KUKA KRL program: Vessel04speedt3.src

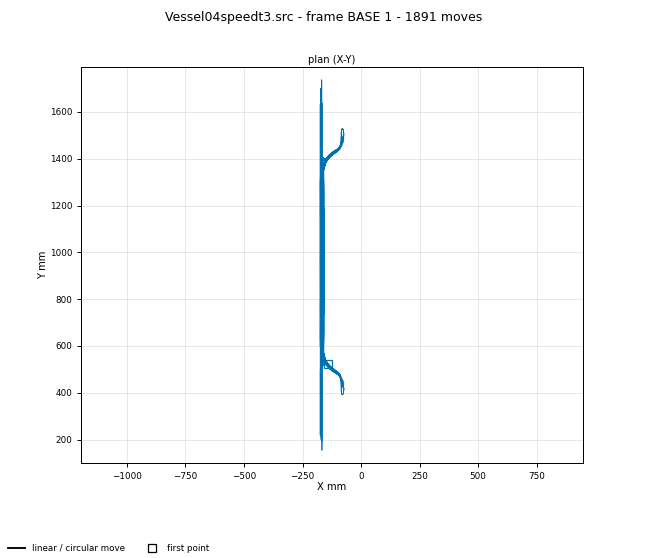
[picture p0: tool path of Vessel04speedt3.src in frame BASE 1, 1891 of 1892 moves have a stored position in this frame; points joined in program order, loops and branches not executed]
&ACCESS RVP
DEF Vessel_04( )
;FOLD INI;%{PE}%V2.2.2,%MKUKATPBASIS,%CINIT,%VCOMMON,%P
;FOLD BAS INI;%{PE}%V2.2.2,%MKUKATPBASIS,%CINIT,%VINIT,%P
INTERRUPT DECL 3 WHEN $STOPMESS==TRUE DO IR_STOPM ( )
INTERRUPT ON 3
BAS (#INITMOV,0 )
;ENDFOLD
;FOLD USER INI;%{P}%V2.2.2,%MKUKATPUSER,%CINIT,%VINIT,%P
;Make your modifications here

;ENDFOLD
;ENDFOLD
ACTION(#AXIS_RESET,34,1000,#NOERROR,ERROR_CODE)
;FOLD PTP HOME  Vel= 100 % DEFAULT;%{PE}%V2.2.2,%MKUKATPBASIS,%CMOVE,%VPTP,%P 1:PTP, 2:HOME, 3:, 5:100, 7:DEFAULT
$H_POS=XHOME
PDAT_ACT=PDEFAULT
BAS (#PTP_DAT )
FDAT_ACT=FHOME
BAS (#FRAMES )
BAS (#VEL_PTP,100 )
PTP  XHOME
;ENDFOLD
BAS(#TOOL,1)
BAS(#BASE,1)
LIN {X -141.371,Y 523.534,Z 0.000,A 30.000, B 0.00, C 0.00,E1 -59.199}
HALT

; PLY 1 OF 41 (Helical)

; ANGLE 51.0 (Not valid for Circ layers and non-tubes)
$APO.CDIS=85
$VEL_EXTAX[1]=100
FOR N_CYC=1 to 56
 LIN_REL {X  -10.568,Y +19.006,A +0.000,E1 -7.240,E3 +6.829,E4 +6.829} C_DIS
 LIN_REL {X  -10.476,Y +36.643,A +0.000,E1 -6.561,E3 +10.073,E4 +10.073} C_DIS
 LIN_REL {X  -2.489,Y +48.216,A -0.000,E1 -2.729,E3 +13.363,E4 +13.363} C_DIS
 LIN_REL {X  +0.199,Y +33.447,A -2.982,E1 -0.404,E3 +10.273,E4 +10.273} C_DIS
 LIN_REL {X  +0.568,Y +37.624,A -7.584,E1 -0.184,E3 +12.184,E4 +12.184} C_DIS
 LIN_REL {X  +1.054,Y +53.527,A -6.791,E1 -0.176,E3 +18.278,E4 +18.278} C_DIS
 LIN_REL {X  +0.629,Y +62.690,A -5.877,E1 +0.690,E3 +22.592,E4 +22.592} C_DIS
 LIN_REL {X  -0.282,Y +46.012,A -4.843,E1 +0.643,E3 +17.284,E4 +17.284} C_DIS
 LIN_REL {X  -0.828,Y +43.828,A -1.901,E1 +0.054,E3 +17.077,E4 +17.077} C_DIS
 LIN_REL {X  -0.963,Y +65.510,A -0.022,E1 -0.470,E3 +27.232,E4 +27.232} C_DIS
 LIN_REL {X  +0.036,Y +73.951,A +0.000,E1 +0.019,E3 +32.052,E4 +32.052} C_DIS
 LIN_REL {X  +0.003,Y +169.509,A +0.000,E1 +0.001,E3 +73.597,E4 +73.597} C_DIS
 LIN_REL {X  +0.150,Y +71.344,A +0.000,E1 +0.017,E3 +31.107,E4 +31.107} C_DIS
 LIN_REL {X  +3.036,Y +57.808,A +0.000,E1 +0.283,E3 +27.550,E4 +27.550} C_DIS
 LIN_REL {X  +11.901,Y +41.351,A +0.000,E1 +1.145,E3 +26.975,E4 +26.975} C_DIS
 LIN_REL {X  +17.652,Y +24.337,A -0.003,E1 +1.971,E3 +20.974,E4 +20.974} C_DIS
 LIN_REL {X  +10.669,Y +8.551,A -2.858,E1 +1.178,E3 +8.021,E4 +8.021} C_DIS
 LIN_REL {X  +17.182,Y +15.853,A -9.749,E1 +3.486,E3 +17.744,E4 +17.744} C_DIS
 LIN_REL {X  +18.322,Y +27.598,A -9.305,E1 +5.329,E3 +37.822,E4 +37.822} C_DIS
 LIN_REL {X  +8.849,Y +21.653,A -6.390,E1 +5.112,E3 +38.276,E4 +38.276} C_DIS
 LIN_REL {X  +4.056,Y +23.007,A -1.638,E1 +5.484,E3 +50.951,E4 +50.951} C_DIS
 LIN_REL {X  -4.096,Y +21.816,A -0.057,E1 +6.652,E3 +66.123,E4 +66.123} C_DIS
 LIN_REL {X  -5.666,Y +0.355,A +0.000,E1 +5.437,E3 +42.648,E4 +42.648} C_DIS
 LIN_REL {X  -2.099,Y -14.454,A +0.000,E1 +6.219,E3 +26.192,E4 +26.192} C_DIS
 LIN_REL {X  -0.280,Y -28.083,A +0.000,E1 +13.715,E3 +25.118,E4 +25.118} C_DIS
 LIN_REL {X  -0.395,Y -28.470,A +0.000,E1 +18.975,E3 +19.603,E4 +19.603} C_DIS
 LIN_REL {X  -9.197,Y -20.928,A +0.000,E1 +22.023,E3 +21.222,E4 +21.222} C_DIS
 LIN_REL {X  -19.997,Y -14.564,A +0.000,E1 +18.453,E3 +20.224,E4 +20.224} C_DIS
 LIN_REL {X  -17.121,Y -13.356,A +0.000,E1 +14.454,E3 +11.101,E4 +11.101} C_DIS
 LIN_REL {X  -9.075,Y -8.563,A +0.000,E1 +4.448,E3 +5.875,E4 +5.875} C_DIS
 LIN_REL {X  -9.764,Y -16.650,A +0.000,E1 +6.452,E3 +6.408,E4 +6.408} C_DIS
 LIN_REL {X  -12.054,Y -40.028,A +0.000,E1 +7.722,E3 +11.062,E4 +11.062} C_DIS
 LIN_REL {X  -2.489,Y -48.280,A +0.000,E1 +2.729,E3 +13.364,E4 +13.364} C_DIS
 LIN_REL {X  +0.199,Y -33.492,A +2.982,E1 +0.404,E3 +10.272,E4 +10.272} C_DIS
 LIN_REL {X  +0.568,Y -37.669,A +7.584,E1 +0.184,E3 +12.184,E4 +12.184} C_DIS
 LIN_REL {X  +1.054,Y -53.586,A +6.791,E1 +0.176,E3 +18.279,E4 +18.279} C_DIS
 LIN_REL {X  +0.629,Y -62.759,A +5.877,E1 -0.690,E3 +22.592,E4 +22.592} C_DIS
 LIN_REL {X  -0.282,Y -46.062,A +4.843,E1 -0.643,E3 +17.283,E4 +17.283} C_DIS
 LIN_REL {X  -0.828,Y -43.872,A +1.901,E1 -0.054,E3 +17.077,E4 +17.077} C_DIS
 LIN_REL {X  -0.963,Y -65.584,A +0.022,E1 +0.470,E3 +27.232,E4 +27.232} C_DIS
 LIN_REL {X  +0.036,Y -74.040,A +0.000,E1 -0.019,E3 +32.053,E4 +32.053} C_DIS
 LIN_REL {X  +0.003,Y -169.741,A +0.000,E1 -0.001,E3 +73.597,E4 +73.597} C_DIS
 LIN_REL {X  +0.150,Y -71.439,A +0.000,E1 -0.017,E3 +31.106,E4 +31.106} C_DIS
 LIN_REL {X  +3.036,Y -57.877,A +0.000,E1 -0.283,E3 +27.551,E4 +27.551} C_DIS
 LIN_REL {X  +11.901,Y -41.410,A +0.000,E1 -1.145,E3 +26.974,E4 +26.974} C_DIS
 LIN_REL {X  +17.652,Y -24.387,A +0.003,E1 -1.971,E3 +20.974,E4 +20.974} C_DIS
 LIN_REL {X  +10.669,Y -8.581,A +2.858,E1 -1.178,E3 +8.021,E4 +8.021} C_DIS
 LIN_REL {X  +17.182,Y -15.882,A +9.749,E1 -3.486,E3 +17.745,E4 +17.745} C_DIS
 LIN_REL {X  +18.322,Y -27.638,A +9.305,E1 -5.329,E3 +37.822,E4 +37.822} C_DIS
 LIN_REL {X  +8.849,Y -21.682,A +6.390,E1 -5.112,E3 +38.276,E4 +38.276} C_DIS
 LIN_REL {X  +4.056,Y -23.042,A +1.638,E1 -5.484,E3 +50.950,E4 +50.950} C_DIS
 LIN_REL {X  -4.096,Y -21.856,A +0.057,E1 -6.652,E3 +66.124,E4 +66.124} C_DIS
 LIN_REL {X  -5.666,Y -0.329,A -0.000,E1 -5.437,E3 +42.647,E4 +42.647} C_DIS
 LIN_REL {X  -2.099,Y +14.582,A -0.000,E1 -6.219,E3 +26.193,E4 +26.193} C_DIS
 LIN_REL {X  -0.280,Y +28.321,A -0.000,E1 -13.715,E3 +25.117,E4 +25.117} C_DIS
 LIN_REL {X  -0.395,Y +28.733,A -0.000,E1 -18.975,E3 +19.604,E4 +19.604} C_DIS
 LIN_REL {X  -9.197,Y +21.087,A -0.000,E1 -22.023,E3 +21.222,E4 +21.222} C_DIS
 LIN_REL {X  -19.997,Y +14.748,A -0.000,E1 -18.452,E3 +20.222,E4 +20.222} C_DIS
 LIN_REL {X  -26.970,Y +23.197,A -0.000,E1 -19.276,E3 +17.546,E4 +17.546} C_DIS
ENDFOR

HALT
LIN {X -165.446,Y 526.668,Z 0.000,A 30.000, B 0.00, C 0.00,E1 -64.562}
HALT

; PLY 2 OF 41 (Connector)

; ANGLE 51.0 (Not valid for Circ layers and non-tubes)
$APO.CDIS=85
$VEL_EXTAX[1]=100
FOR N_CYC=1 to 1
 LIN_REL {X  +0.000,Y +6.669,A +0.000,E1 -1.453,E3 +1.289,E4 +1.289} C_DIS
 LIN_REL {X  +0.000,Y +15.761,A +0.000,E1 -3.190,E3 +3.934,E4 +3.934} C_DIS
 LIN_REL {X  +0.000,Y +31.342,A +0.000,E1 -3.400,E3 +9.789,E4 +9.789} C_DIS
 LIN_REL {X  +0.000,Y +43.799,A +0.000,E1 -1.567,E3 +14.926,E4 +14.926} C_DIS
 LIN_REL {X  +0.000,Y +28.255,A -1.983,E1 -0.087,E3 +10.643,E4 +10.643} C_DIS
 LIN_REL {X  +0.000,Y +29.952,A -7.476,E1 +0.318,E3 +11.872,E4 +11.872} C_DIS
 LIN_REL {X  +0.000,Y +47.685,A -7.690,E1 +0.225,E3 +20.095,E4 +20.095} C_DIS
 LIN_REL {X  +0.000,Y +55.129,A -7.422,E1 +0.668,E3 +25.472,E4 +25.472} C_DIS
 LIN_REL {X  +0.000,Y +43.863,A -4.702,E1 +1.177,E3 +22.727,E4 +22.727} C_DIS
 LIN_REL {X  +0.000,Y +50.043,A -0.726,E1 +1.544,E3 +40.796,E4 +40.796} C_DIS
 LIN_REL {X  +0.000,Y +46.945,A -0.001,E1 +3.695,E3 +57.103,E4 +57.103} C_DIS
 LIN_REL {X  +0.000,Y +58.316,A +0.000,E1 +4.226,E3 +72.975,E4 +72.975} C_DIS
 LIN_REL {X  +0.000,Y +65.060,A +0.000,E1 +4.740,E3 +89.502,E4 +89.502} C_DIS
 LIN_REL {X  +0.000,Y +67.059,A +0.000,E1 +5.237,E3 +105.894,E4 +105.894} C_DIS
 LIN_REL {X  +0.000,Y +54.897,A +0.000,E1 +4.784,E3 +101.231,E4 +101.231} C_DIS
 LIN_REL {X  +0.000,Y +40.560,A +0.000,E1 +3.986,E3 +86.611,E4 +86.611} C_DIS
 LIN_REL {X  +0.000,Y +28.994,A +0.000,E1 +3.229,E3 +70.429,E4 +70.429} C_DIS
 LIN_REL {X  +0.000,Y +20.924,A -0.000,E1 +3.270,E3 +56.833,E4 +56.833} C_DIS
 LIN_REL {X  +0.000,Y +10.940,A -0.000,E1 +2.663,E3 +31.936,E4 +31.936} C_DIS
 LIN_REL {X  +0.000,Y +9.716,A -0.000,E1 +1.163,E3 +31.606,E4 +31.606} C_DIS
 LIN_REL {X  +0.000,Y +17.235,A -0.000,E1 +1.953,E3 +55.180,E4 +55.180} C_DIS
 LIN_REL {X  +0.000,Y +19.045,A -0.003,E1 +3.492,E3 +73.663,E4 +73.663} C_DIS
 LIN_REL {X  +0.000,Y +14.681,A -0.050,E1 +3.224,E3 +66.879,E4 +66.879} C_DIS
 LIN_REL {X  +0.000,Y +9.269,A -0.348,E1 +2.308,E3 +46.823,E4 +46.823} C_DIS
 LIN_REL {X  +0.000,Y +6.944,A -1.216,E1 +1.589,E3 +34.534,E4 +34.534} C_DIS
 LIN_REL {X  +0.000,Y +4.516,A -2.642,E1 +2.440,E3 +22.764,E4 +22.764} C_DIS
 LIN_REL {X  +0.000,Y +6.499,A -8.076,E1 +7.847,E3 +36.933,E4 +36.933} C_DIS
 LIN_REL {X  +0.000,Y +2.636,A -11.608,E1 +16.156,E3 +54.770,E4 +54.770} C_DIS
 LIN_REL {X  +0.000,Y -5.220,A -5.677,E1 +11.730,E3 +42.954,E4 +42.954} C_DIS
 LIN_REL {X  +0.000,Y -8.791,A -0.380,E1 +8.530,E3 +42.436,E4 +42.436} C_DIS
 LIN_REL {X  +0.000,Y -12.212,A +0.684,E1 +4.305,E3 +49.511,E4 +49.511} C_DIS
 LIN_REL {X  +0.000,Y -10.625,A +3.317,E1 +0.257,E3 +39.510,E4 +39.510} C_DIS
 LIN_REL {X  +0.000,Y -13.460,A +7.461,E1 -1.466,E3 +45.445,E4 +45.445} C_DIS
 LIN_REL {X  +0.000,Y -11.035,A +8.147,E1 -3.492,E3 +45.926,E4 +45.926} C_DIS
 LIN_REL {X  +0.000,Y -5.827,A +5.802,E1 -4.151,E3 +33.734,E4 +33.734} C_DIS
 LIN_REL {X  +0.000,Y -3.469,A +3.163,E1 -3.757,E3 +23.171,E4 +23.171} C_DIS
 LIN_REL {X  +0.000,Y -3.190,A +0.984,E1 -1.508,E3 +21.680,E4 +21.680} C_DIS
 LIN_REL {X  +0.000,Y -7.110,A +0.259,E1 -0.070,E3 +43.916,E4 +43.916} C_DIS
 LIN_REL {X  +0.000,Y -11.368,A +0.138,E1 -0.176,E3 +67.863,E4 +67.863} C_DIS
 LIN_REL {X  +0.000,Y -14.551,A +0.038,E1 -0.171,E3 +86.686,E4 +86.686} C_DIS
 LIN_REL {X  +0.000,Y -18.070,A +0.007,E1 -0.196,E3 +109.624,E4 +109.624} C_DIS
 LIN_REL {X  +0.000,Y -22.012,A -0.000,E1 -0.254,E3 +135.858,E4 +135.858} C_DIS
 LIN_REL {X  +0.000,Y -21.223,A -0.000,E1 -0.248,E3 +133.245,E4 +133.245} C_DIS
 LIN_REL {X  +0.000,Y -21.216,A +0.000,E1 -0.253,E3 +135.616,E4 +135.616} C_DIS
 LIN_REL {X  +0.000,Y -19.639,A +0.000,E1 -0.238,E3 +127.722,E4 +127.722} C_DIS
 LIN_REL {X  +0.000,Y -22.775,A +0.000,E1 -0.282,E3 +150.992,E4 +150.992} C_DIS
 LIN_REL {X  +0.000,Y -19.627,A +0.000,E1 -0.247,E3 +132.648,E4 +132.648} C_DIS
 LIN_REL {X  +0.000,Y -18.051,A +0.000,E1 -0.232,E3 +124.267,E4 +124.267} C_DIS
 LIN_REL {X  +0.000,Y -16.360,A +0.000,E1 -0.240,E3 +115.340,E4 +115.340} C_DIS
 LIN_REL {X  +0.000,Y -13.190,A +0.000,E1 -0.197,E3 +93.494,E4 +93.494} C_DIS
 LIN_REL {X  +0.000,Y -18.226,A +0.000,E1 -0.208,E3 +131.179,E4 +131.179} C_DIS
 LIN_REL {X  +0.000,Y -18.142,A +0.000,E1 -0.250,E3 +133.669,E4 +133.669} C_DIS
 LIN_REL {X  +0.000,Y -16.791,A +0.000,E1 -0.236,E3 +126.245,E4 +126.245} C_DIS
 LIN_REL {X  +0.000,Y -17.456,A +0.000,E1 -0.251,E3 +133.939,E4 +133.939} C_DIS
 LIN_REL {X  +0.000,Y -18.120,A +0.000,E1 -0.266,E3 +142.029,E4 +142.029} C_DIS
 LIN_REL {X  +0.000,Y -16.100,A +0.000,E1 -0.241,E3 +128.959,E4 +128.959} C_DIS
 LIN_REL {X  +0.000,Y -13.909,A +0.000,E1 -0.253,E3 +114.655,E4 +114.655} C_DIS
 LIN_REL {X  +0.000,Y -13.331,A +0.000,E1 -0.189,E3 +110.307,E4 +110.307} C_DIS
 LIN_REL {X  +0.000,Y -14.682,A +0.000,E1 -0.222,E3 +124.521,E4 +124.521} C_DIS
 LIN_REL {X  +0.000,Y -14.649,A +0.000,E1 -0.238,E3 +127.210,E4 +127.210} C_DIS
 LIN_REL {X  +0.000,Y -14.642,A +0.000,E1 -0.245,E3 +130.081,E4 +130.081} C_DIS
 LIN_REL {X  +0.000,Y -14.049,A +0.000,E1 -0.240,E3 +127.771,E4 +127.771} C_DIS
 LIN_REL {X  +0.000,Y -13.316,A +0.000,E1 -0.266,E3 +124.898,E4 +124.898} C_DIS
 LIN_REL {X  +0.000,Y -12.811,A +0.000,E1 -0.214,E3 +121.425,E4 +121.425} C_DIS
 LIN_REL {X  +0.000,Y -13.525,A +0.000,E1 -0.239,E3 +131.925,E4 +131.925} C_DIS
 LIN_REL {X  +0.000,Y -13.496,A +0.000,E1 -0.255,E3 +135.380,E4 +135.380} C_DIS
 LIN_REL {X  +0.000,Y -13.916,A +0.000,E1 -0.292,E3 +144.481,E4 +144.481} C_DIS
 LIN_REL {X  +0.000,Y -15.433,A +0.000,E1 -0.302,E3 +163.677,E4 +163.677} C_DIS
 LIN_REL {X  +0.000,Y -13.062,A +0.000,E1 -0.265,E3 +143.836,E4 +143.836} C_DIS
 LIN_REL {X  +0.000,Y -14.351,A +0.000,E1 -0.330,E3 +164.500,E4 +164.500} C_DIS
 LIN_REL {X  +0.000,Y -14.752,A +0.000,E1 -0.322,E3 +174.175,E4 +174.175} C_DIS
 LIN_REL {X  +0.000,Y -13.520,A +0.000,E1 -0.312,E3 +167.011,E4 +167.011} C_DIS
 LIN_REL {X  +0.000,Y -14.261,A +0.000,E1 -0.368,E3 +185.009,E4 +185.009} C_DIS
 LIN_REL {X  +0.000,Y -13.726,A +0.000,E1 -0.362,E3 +186.241,E4 +186.241} C_DIS
 LIN_REL {X  +0.000,Y -14.142,A +0.000,E1 -0.375,E3 +201.491,E4 +201.491} C_DIS
 LIN_REL {X  +0.000,Y -16.249,A +0.000,E1 -0.488,E3 +248.169,E4 +248.169} C_DIS
 LIN_REL {X  +0.000,Y -13.146,A +0.000,E1 -0.419,E3 +216.296,E4 +216.296} C_DIS
 LIN_REL {X  +0.000,Y -12.536,A +0.000,E1 -0.444,E3 +223.007,E4 +223.007} C_DIS
 LIN_REL {X  +0.000,Y -13.931,A +0.002,E1 -0.528,E3 +269.089,E4 +269.089} C_DIS
 LIN_REL {X  +0.000,Y -14.238,A +0.015,E1 -0.664,E3 +311.059,E4 +311.059} C_DIS
 LIN_REL {X  +0.000,Y -12.921,A +0.080,E1 -0.909,E3 +334.214,E4 +334.214} C_DIS
 LIN_REL {X  +0.000,Y -8.261,A +0.329,E1 -2.001,E3 +312.120,E4 +312.120} C_DIS
 LIN_REL {X  +0.000,Y -2.591,A +0.480,E1 -1.840,E3 +356.413,E4 +356.413} C_DIS
 LIN_REL {X  +0.000,Y -0.100,A +0.024,E1 -0.087,E3 +16.643,E4 +16.643} C_DIS
ENDFOR

HALT
LIN {X -165.446,Y 600.000,Z 0.000,A 0.000, B 0.00, C 0.00,E1 -0.000}
HALT

; PLY 3 OF 41 (Circ)

; ANGLE 51.0 (Not valid for Circ layers and non-tubes)
$APO.CDIS=85
$VEL_EXTAX[1]=100
FOR N_CYC=1 to 1
 LIN_REL {X  +0.000,Y +0.000,A +0.000,E1 +0.000,E3 +13.889,E4 +13.889} C_DIS
 LIN_REL {X  +0.000,Y +6.750,A +0.000,E1 -0.981,E3 +500.000,E4 +500.000} C_DIS
 LIN_REL {X  +0.000,Y +706.500,A +0.000,E1 -0.000,E3 +52333.333,E4 +52333.333} C_DIS
 LIN_REL {X  +0.000,Y +6.750,A +0.000,E1 +0.981,E3 +500.000,E4 +500.000} C_DIS
 LIN_REL {X  +0.000,Y +0.000,A +0.000,E1 +0.000,E3 +500.000,E4 +500.000} C_DIS
 LIN_REL {X  +0.000,Y -6.750,A +0.000,E1 +0.981,E3 +500.000,E4 +500.000} C_DIS
 LIN_REL {X  +0.000,Y -706.500,A +0.000,E1 +0.000,E3 +52333.334,E4 +52333.334} C_DIS
 LIN_REL {X  +0.000,Y -6.750,A +0.000,E1 -0.981,E3 +500.000,E4 +500.000} C_DIS
 LIN_REL {X  +0.000,Y +0.000,A +0.000,E1 +0.000,E3 +13.889,E4 +13.889} C_DIS
ENDFOR

HALT
LIN {X -165.150,Y 600.770,Z 0.000,A 6.131, B 0.00, C 0.00,E1 -8.082}
HALT

; PLY 4 OF 41 (Helical)

; ANGLE 51.0 (Not valid for Circ layers and non-tubes)
$APO.CDIS=85
$VEL_EXTAX[1]=100
FOR N_CYC=1 to 7
 LIN_REL {X  +1.504,Y +4.220,A -1.773,E1 -0.081,E3 +55.957,E4 +55.957} C_DIS
 LIN_REL {X  +0.876,Y +6.465,A -2.206,E1 -0.007,E3 +72.171,E4 +72.171} C_DIS
 LIN_REL {X  +0.141,Y +8.567,A -1.722,E1 +0.003,E3 +86.313,E4 +86.313} C_DIS
 LIN_REL {X  +0.163,Y +8.806,A -0.396,E1 +0.019,E3 +101.457,E4 +101.457} C_DIS
 LIN_REL {X  -0.118,Y +10.236,A -0.013,E1 +0.019,E3 +123.687,E4 +123.687} C_DIS
 LIN_REL {X  -0.093,Y +16.128,A -0.020,E1 +0.021,E3 +194.227,E4 +194.227} C_DIS
 LIN_REL {X  +0.004,Y +631.468,A -0.003,E1 +0.005,E3 +7614.921,E4 +7614.921} C_DIS
 LIN_REL {X  +0.137,Y +12.187,A -0.021,E1 +0.014,E3 +146.411,E4 +146.411} C_DIS
 LIN_REL {X  +0.398,Y +16.778,A +0.064,E1 -0.045,E3 +203.049,E4 +203.049} C_DIS
 LIN_REL {X  +0.295,Y +7.687,A -0.774,E1 +1.054,E3 +101.508,E4 +101.508} C_DIS
 LIN_REL {X  +0.019,Y +4.371,A -1.638,E1 +2.222,E3 +73.577,E4 +73.577} C_DIS
 LIN_REL {X  -0.436,Y +0.938,A -3.346,E1 +5.266,E3 +73.263,E4 +73.263} C_DIS
 LIN_REL {X  -0.504,Y -3.799,A -2.772,E1 +6.377,E3 +53.588,E4 +53.588} C_DIS
 LIN_REL {X  -0.171,Y -5.172,A +1.553,E1 +2.247,E3 +39.654,E4 +39.654} C_DIS
 LIN_REL {X  +0.174,Y -7.524,A +3.099,E1 +0.473,E3 +61.006,E4 +61.006} C_DIS
 LIN_REL {X  +0.244,Y -7.265,A +3.270,E1 -1.468,E3 +71.734,E4 +71.734} C_DIS
 LIN_REL {X  +0.047,Y -7.571,A +0.620,E1 -0.115,E3 +85.531,E4 +85.531} C_DIS
 LIN_REL {X  -0.078,Y -12.227,A -0.079,E1 +0.215,E3 +145.433,E4 +145.433} C_DIS
 LIN_REL {X  -0.090,Y -11.440,A +0.014,E1 -0.018,E3 +137.818,E4 +137.818} C_DIS
 LIN_REL {X  -0.026,Y -640.154,A +0.014,E1 -0.016,E3 +7719.473,E4 +7719.473} C_DIS
 LIN_REL {X  +0.150,Y -12.185,A +0.021,E1 -0.014,E3 +146.397,E4 +146.397} C_DIS
 LIN_REL {X  +0.423,Y -16.780,A +0.233,E1 -0.216,E3 +203.108,E4 +203.108} C_DIS
 LIN_REL {X  +0.049,Y -6.526,A +0.791,E1 -1.151,E3 +90.121,E4 +90.121} C_DIS
 LIN_REL {X  -0.013,Y -4.018,A +1.149,E1 -2.020,E3 +70.590,E4 +70.590} C_DIS
 LIN_REL {X  -0.254,Y -0.953,A +2.186,E1 -4.682,E3 +73.216,E4 +73.216} C_DIS
 LIN_REL {X  -2.061,Y +5.137,A +1.321,E1 -5.684,E3 +59.531,E4 +59.531} C_DIS
 LIN_REL {X  -0.780,Y +2.626,A +0.428,E1 -2.418,E3 +53.402,E4 +53.402} C_DIS
ENDFOR

HALT
LIN {X -166.522,Y 598.723,Z 0.000,A 0.303, B 0.00, C 0.00,E1 -1.645}
HALT

; PLY 5 OF 41 (Connector)

; ANGLE 51.0 (Not valid for Circ layers and non-tubes)
$APO.CDIS=85
$VEL_EXTAX[1]=100
FOR N_CYC=1 to 1
 LIN_REL {X  +0.000,Y +1.277,A -0.000,E1 +1.385,E3 +231.040,E4 +231.040} C_DIS
ENDFOR

HALT
LIN {X -166.524,Y 600.000,Z 0.000,A 0.000, B 0.00, C 0.00,E1 -0.000}
HALT

; PLY 6 OF 41 (Circ)

; ANGLE 51.0 (Not valid for Circ layers and non-tubes)
$APO.CDIS=85
$VEL_EXTAX[1]=100
FOR N_CYC=1 to 1
 LIN_REL {X  +0.000,Y +1.277,A -0.000,E1 +1.385,E3 +231.040,E4 +231.040} C_DIS
 LIN_REL {X  +0.000,Y +6.750,A -0.000,E1 -0.973,E3 +500.000,E4 +500.000} C_DIS
 LIN_REL {X  +0.000,Y +706.500,A -0.000,E1 +0.000,E3 +52333.333,E4 +52333.333} C_DIS
 LIN_REL {X  +0.000,Y +6.750,A -0.000,E1 +0.973,E3 +500.000,E4 +500.000} C_DIS
 LIN_REL {X  +0.000,Y +0.000,A -0.000,E1 -0.000,E3 +500.000,E4 +500.000} C_DIS
 LIN_REL {X  +0.000,Y -6.750,A -0.000,E1 +0.973,E3 +500.000,E4 +500.000} C_DIS
 LIN_REL {X  +0.000,Y -706.500,A -0.000,E1 -0.000,E3 +52333.333,E4 +52333.333} C_DIS
 LIN_REL {X  +0.000,Y -6.750,A -0.000,E1 -0.973,E3 +500.000,E4 +500.000} C_DIS
 LIN_REL {X  +0.000,Y +0.000,A -0.000,E1 -0.000,E3 +13.889,E4 +13.889} C_DIS
ENDFOR

HALT
LIN {X -166.866,Y 600.000,Z 0.000,A 2.748, B 0.00, C 0.00,E1 -2.357}
HALT

; PLY 7 OF 41 (Connector)

; ANGLE 51.0 (Not valid for Circ layers and non-tubes)
$APO.CDIS=85
$VEL_EXTAX[1]=100
FOR N_CYC=1 to 1
 LIN_REL {X  +0.000,Y +2.709,A -0.375,E1 -1.968,E3 +22.875,E4 +22.875} C_DIS
 LIN_REL {X  +0.000,Y +5.934,A -1.379,E1 -2.655,E3 +43.522,E4 +43.522} C_DIS
 LIN_REL {X  +0.000,Y +8.070,A -0.851,E1 -2.120,E3 +63.008,E4 +63.008} C_DIS
 LIN_REL {X  +0.000,Y +13.115,A -0.322,E1 -3.320,E3 +80.297,E4 +80.297} C_DIS
 LIN_REL {X  +0.000,Y +20.471,A +0.186,E1 -4.390,E3 +96.984,E4 +96.984} C_DIS
 LIN_REL {X  +0.000,Y +24.441,A -0.001,E1 -4.109,E3 +92.330,E4 +92.330} C_DIS
 LIN_REL {X  +0.000,Y +28.284,A -0.006,E1 -3.844,E3 +87.285,E4 +87.285} C_DIS
 LIN_REL {X  +0.000,Y +25.603,A -0.000,E1 -3.033,E3 +69.707,E4 +69.707} C_DIS
 LIN_REL {X  +0.000,Y +30.257,A -0.000,E1 -3.222,E3 +72.218,E4 +72.218} C_DIS
 LIN_REL {X  +0.000,Y +28.011,A -0.000,E1 -2.715,E3 +59.690,E4 +59.690} C_DIS
 LIN_REL {X  +0.000,Y +21.466,A -0.000,E1 -1.989,E3 +40.385,E4 +40.385} C_DIS
 LIN_REL {X  +0.000,Y +19.564,A -0.000,E1 -1.787,E3 +35.011,E4 +35.011} C_DIS
 LIN_REL {X  +0.000,Y +14.769,A -0.000,E1 -0.876,E3 +27.909,E4 +27.909} C_DIS
 LIN_REL {X  +0.000,Y +21.828,A -0.000,E1 -1.310,E3 +36.234,E4 +36.234} C_DIS
 LIN_REL {X  +0.000,Y +32.021,A -0.000,E1 -2.261,E3 +49.976,E4 +49.976} C_DIS
 LIN_REL {X  +0.000,Y +44.064,A -0.000,E1 -2.932,E3 +62.790,E4 +62.790} C_DIS
 LIN_REL {X  +0.000,Y +57.726,A -0.000,E1 -3.466,E3 +73.369,E4 +73.369} C_DIS
 LIN_REL {X  +0.000,Y +74.702,A -0.000,E1 -3.987,E3 +82.699,E4 +82.699} C_DIS
 LIN_REL {X  +0.000,Y +79.300,A -0.000,E1 -3.747,E3 +75.342,E4 +75.342} C_DIS
 LIN_REL {X  +0.000,Y +84.555,A -0.000,E1 -3.560,E3 +68.621,E4 +68.621} C_DIS
 LIN_REL {X  +0.000,Y +90.749,A -0.000,E1 -3.413,E3 +62.266,E4 +62.266} C_DIS
 LIN_REL {X  +0.000,Y +82.276,A -0.001,E1 -2.787,E3 +47.674,E4 +47.674} C_DIS
 LIN_REL {X  +0.000,Y +68.384,A -0.015,E1 -2.115,E3 +34.134,E4 +34.134} C_DIS
 LIN_REL {X  +0.000,Y +48.811,A -0.666,E1 -1.358,E3 +22.878,E4 +22.878} C_DIS
 LIN_REL {X  +0.000,Y +28.049,A -0.431,E1 -0.487,E3 +15.828,E4 +15.828} C_DIS
 LIN_REL {X  +0.000,Y +24.580,A -4.555,E1 -1.342,E3 +21.887,E4 +21.887} C_DIS
 LIN_REL {X  +0.000,Y +26.318,A -13.544,E1 +4.685,E3 +36.180,E4 +36.180} C_DIS
 LIN_REL {X  +0.000,Y +12.666,A -9.119,E1 +4.744,E3 +27.176,E4 +27.176} C_DIS
 LIN_REL {X  +0.000,Y +9.587,A -1.669,E1 +10.874,E3 +38.750,E4 +38.750} C_DIS
 LIN_REL {X  +0.000,Y +2.443,A -0.000,E1 +5.402,E3 +14.033,E4 +14.033} C_DIS
 LIN_REL {X  +0.000,Y +2.065,A -0.000,E1 -0.441,E3 +8.789,E4 +8.789} C_DIS
 LIN_REL {X  +0.000,Y +3.157,A -0.000,E1 -10.062,E3 +4.975,E4 +4.975} C_DIS
 LIN_REL {X  +0.000,Y +1.720,A -0.000,E1 -0.635,E3 +6.845,E4 +6.845} C_DIS
 LIN_REL {X  +0.000,Y -13.023,A -0.000,E1 +6.086,E3 +22.111,E4 +22.111} C_DIS
 LIN_REL {X  +0.000,Y -38.062,A -0.000,E1 +9.514,E3 +32.445,E4 +32.445} C_DIS
 LIN_REL {X  +0.000,Y -44.509,A -0.000,E1 +17.078,E3 +26.528,E4 +26.528} C_DIS
 LIN_REL {X  +0.000,Y -33.762,A -0.000,E1 +19.289,E3 +16.182,E4 +16.182} C_DIS
 LIN_REL {X  +0.000,Y -27.705,A -0.000,E1 +18.648,E3 +11.508,E4 +11.508} C_DIS
 LIN_REL {X  +0.000,Y -30.449,A -0.000,E1 +19.082,E3 +11.153,E4 +11.153} C_DIS
 LIN_REL {X  +0.000,Y -28.699,A -0.000,E1 +14.042,E3 +9.805,E4 +9.805} C_DIS
 LIN_REL {X  +0.000,Y -15.614,A -0.000,E1 +6.102,E3 +5.459,E4 +5.459} C_DIS
 LIN_REL {X  +0.000,Y -14.684,A -0.000,E1 +4.349,E3 +4.700,E4 +4.700} C_DIS
 LIN_REL {X  +0.000,Y -18.247,A -0.000,E1 +4.966,E3 +4.318,E4 +4.318} C_DIS
 LIN_REL {X  +0.000,Y -40.805,A -0.000,E1 +6.873,E3 +9.579,E4 +9.579} C_DIS
 LIN_REL {X  +0.000,Y -43.385,A -0.000,E1 +2.911,E3 +13.389,E4 +13.389} C_DIS
 LIN_REL {X  +0.000,Y -21.697,A +1.407,E1 +0.491,E3 +7.414,E4 +7.414} C_DIS
 LIN_REL {X  +0.000,Y -15.906,A +3.938,E1 +0.128,E3 +5.509,E4 +5.509} C_DIS
 LIN_REL {X  +0.000,Y -15.553,A -3.400,E1 +1.586,E3 +5.570,E4 +5.570} C_DIS
 LIN_REL {X  +0.000,Y -26.286,A +1.138,E1 +0.916,E3 +9.871,E4 +9.871} C_DIS
 LIN_REL {X  +0.000,Y -34.188,A +9.795,E1 -1.013,E3 +13.279,E4 +13.279} C_DIS
 LIN_REL {X  +0.000,Y -46.284,A +10.757,E1 -1.729,E3 +18.381,E4 +18.381} C_DIS
 LIN_REL {X  +0.000,Y -40.303,A +4.905,E1 -0.042,E3 +16.060,E4 +16.060} C_DIS
 LIN_REL {X  +0.000,Y -40.789,A +0.215,E1 +1.044,E3 +16.316,E4 +16.316} C_DIS
 LIN_REL {X  +0.000,Y -58.705,A +1.227,E1 +0.105,E3 +25.483,E4 +25.483} C_DIS
 LIN_REL {X  +0.000,Y -68.112,A +0.018,E1 +0.171,E3 +30.702,E4 +30.702} C_DIS
 LIN_REL {X  +0.000,Y -83.645,A -0.000,E1 +0.218,E3 +37.199,E4 +37.199} C_DIS
 LIN_REL {X  +0.000,Y -95.177,A -0.000,E1 +0.246,E3 +41.622,E4 +41.622} C_DIS
 LIN_REL {X  +0.000,Y -95.313,A -0.000,E1 +0.246,E3 +40.935,E4 +40.935} C_DIS
 LIN_REL {X  +0.000,Y -95.451,A -0.000,E1 +0.244,E3 +40.251,E4 +40.251} C_DIS
 LIN_REL {X  +0.000,Y -95.603,A -0.000,E1 +0.244,E3 +39.572,E4 +39.572} C_DIS
 LIN_REL {X  +0.000,Y -88.071,A -0.000,E1 +0.223,E3 +35.801,E4 +35.801} C_DIS
 LIN_REL {X  +0.000,Y -71.311,A -0.038,E1 +0.310,E3 +28.903,E4 +28.903} C_DIS
 LIN_REL {X  +0.000,Y -54.067,A +1.000,E1 +0.485,E3 +26.757,E4 +26.757} C_DIS
 LIN_REL {X  +0.000,Y -37.551,A +3.500,E1 -0.175,E3 +25.576,E4 +25.576} C_DIS
 LIN_REL {X  +0.000,Y -23.752,A +6.225,E1 -1.006,E3 +22.383,E4 +22.383} C_DIS
 LIN_REL {X  +0.000,Y -14.617,A +10.471,E1 -1.579,E3 +21.867,E4 +21.867} C_DIS
 LIN_REL {X  +0.000,Y -6.257,A +4.467,E1 -1.274,E3 +13.799,E4 +13.799} C_DIS
 LIN_REL {X  +0.000,Y -5.913,A +3.889,E1 -6.406,E3 +39.133,E4 +39.133} C_DIS
 LIN_REL {X  +0.000,Y +1.606,A +0.433,E1 -5.272,E3 +19.812,E4 +19.812} C_DIS
 LIN_REL {X  +0.000,Y +3.074,A +0.052,E1 -0.302,E3 +14.777,E4 +14.777} C_DIS
 LIN_REL {X  +0.000,Y +5.841,A +0.001,E1 +6.938,E3 +13.700,E4 +13.700} C_DIS
 LIN_REL {X  +0.000,Y +9.970,A -0.000,E1 -0.096,E3 +11.036,E4 +11.036} C_DIS
 LIN_REL {X  +0.000,Y +32.797,A -0.000,E1 -4.991,E3 +21.247,E4 +21.247} C_DIS
 LIN_REL {X  +0.000,Y +59.430,A -0.000,E1 -7.758,E3 +28.817,E4 +28.817} C_DIS
 LIN_REL {X  +0.000,Y +53.062,A -0.000,E1 -9.132,E3 +20.142,E4 +20.142} C_DIS
 LIN_REL {X  +0.000,Y +45.633,A -0.000,E1 -17.612,E3 +14.654,E4 +14.654} C_DIS
 LIN_REL {X  +0.000,Y +33.155,A -0.000,E1 -21.448,E3 +9.492,E4 +9.492} C_DIS
 LIN_REL {X  +0.000,Y +26.803,A -0.000,E1 -21.163,E3 +7.012,E4 +7.012} C_DIS
 LIN_REL {X  +0.000,Y +28.096,A -0.000,E1 -20.476,E3 +6.712,E4 +6.712} C_DIS
 LIN_REL {X  +0.000,Y +24.825,A -0.000,E1 -13.159,E3 +5.522,E4 +5.522} C_DIS
 LIN_REL {X  +0.000,Y +23.696,A -0.000,E1 -9.477,E3 +4.462,E4 +4.462} C_DIS
 LIN_REL {X  +0.000,Y +13.874,A -0.000,E1 -3.970,E3 +2.183,E4 +2.183} C_DIS
ENDFOR

HALT
LIN {X -143.180,Y 524.782,Z 0.000,A 30.000, B 0.00, C 0.00,E1 -60.639}
HALT

; PLY 8 OF 41 (Helical)

; ANGLE 51.0 (Not valid for Circ layers and non-tubes)
$APO.CDIS=85
$VEL_EXTAX[1]=100
FOR N_CYC=1 to 56
 LIN_REL {X  -11.203,Y +20.731,A +0.000,E1 -6.867,E3 +9.241,E4 +9.241} C_DIS
 LIN_REL {X  -10.898,Y +42.129,A +0.000,E1 -6.326,E3 +12.284,E4 +12.284} C_DIS
 LIN_REL {X  -1.482,Y +42.709,A +0.000,E1 -1.937,E3 +11.913,E4 +11.913} C_DIS
 LIN_REL {X  +0.094,Y +26.249,A -2.547,E1 -0.194,E3 +7.968,E4 +7.968} C_DIS
 LIN_REL {X  +0.269,Y +20.359,A -5.014,E1 -0.020,E3 +6.425,E4 +6.425} C_DIS
 LIN_REL {X  +0.667,Y +27.301,A -0.271,E1 -0.990,E3 +8.885,E4 +8.885} C_DIS
 LIN_REL {X  +0.898,Y +36.715,A -6.122,E1 -0.053,E3 +12.310,E4 +12.310} C_DIS
 LIN_REL {X  +0.530,Y +32.807,A -6.227,E1 +0.829,E3 +11.282,E4 +11.282} C_DIS
 LIN_REL {X  +0.179,Y +44.045,A -3.970,E1 +0.652,E3 +15.551,E4 +15.551} C_DIS
 LIN_REL {X  -0.716,Y +62.764,A -4.463,E1 +0.316,E3 +23.010,E4 +23.010} C_DIS
 LIN_REL {X  -1.437,Y +77.421,A -1.378,E1 -0.313,E3 +30.586,E4 +30.586} C_DIS
 LIN_REL {X  -0.058,Y +90.486,A -0.008,E1 -0.076,E3 +38.244,E4 +38.244} C_DIS
 LIN_REL {X  +0.007,Y +165.811,A +0.000,E1 +0.003,E3 +70.391,E4 +70.391} C_DIS
 LIN_REL {X  +0.070,Y +60.938,A +0.000,E1 +0.008,E3 +25.931,E4 +25.931} C_DIS
 LIN_REL {X  +0.881,Y +43.756,A +0.000,E1 +0.084,E3 +19.277,E4 +19.277} C_DIS
 LIN_REL {X  +3.154,Y +30.505,A +0.000,E1 +0.288,E3 +15.437,E4 +15.437} C_DIS
 LIN_REL {X  +3.138,Y +13.469,A +0.000,E1 +0.286,E3 +8.142,E4 +8.142} C_DIS
 LIN_REL {X  +10.398,Y +24.310,A -0.000,E1 +1.013,E3 +17.741,E4 +17.741} C_DIS
 LIN_REL {X  +18.417,Y +23.422,A -0.344,E1 +2.019,E3 +19.767,E4 +19.767} C_DIS
 LIN_REL {X  +16.730,Y +12.634,A -5.197,E1 +2.228,E3 +13.321,E4 +13.321} C_DIS
 LIN_REL {X  +14.171,Y +12.777,A -10.743,E1 +4.501,E3 +16.589,E4 +16.589} C_DIS
 LIN_REL {X  +12.524,Y +17.798,A -5.333,E1 +4.096,E3 +25.559,E4 +25.559} C_DIS
 LIN_REL {X  +9.943,Y +23.830,A -6.362,E1 +3.953,E3 +40.201,E4 +40.201} C_DIS
 LIN_REL {X  +3.598,Y +17.979,A -1.831,E1 +3.568,E3 +36.484,E4 +36.484} C_DIS
 LIN_REL {X  -1.086,Y +24.134,A -0.190,E1 +5.885,E3 +60.191,E4 +60.191} C_DIS
 LIN_REL {X  -4.618,Y +9.202,A +0.000,E1 +4.719,E3 +40.160,E4 +40.160} C_DIS
 LIN_REL {X  -3.238,Y -2.186,A +0.000,E1 +3.481,E3 +25.337,E4 +25.337} C_DIS
 LIN_REL {X  -2.104,Y -17.155,A +0.000,E1 +7.479,E3 +29.747,E4 +29.747} C_DIS
 LIN_REL {X  -0.218,Y -30.303,A +0.000,E1 +15.565,E3 +26.473,E4 +26.473} C_DIS
 LIN_REL {X  -1.126,Y -27.146,A +0.000,E1 +19.493,E3 +19.475,E4 +19.475} C_DIS
 LIN_REL {X  -10.383,Y -17.338,A +0.000,E1 +20.083,E3 +20.854,E4 +20.854} C_DIS
 LIN_REL {X  -20.496,Y -14.001,A +0.000,E1 +19.322,E3 +20.764,E4 +20.764} C_DIS
 LIN_REL {X  -22.719,Y -19.698,A +0.000,E1 +15.924,E3 +16.964,E4 +16.964} C_DIS
 LIN_REL {X  -18.416,Y -32.580,A +0.000,E1 +10.756,E3 +14.079,E4 +14.079} C_DIS
 LIN_REL {X  -8.146,Y -38.962,A +0.000,E1 +5.009,E3 +10.936,E4 +10.936} C_DIS
 LIN_REL {X  -0.894,Y -42.157,A +0.001,E1 +1.701,E3 +11.815,E4 +11.815} C_DIS
 LIN_REL {X  +0.129,Y -26.139,A +3.688,E1 +0.037,E3 +7.999,E4 +7.999} C_DIS
 LIN_REL {X  +0.308,Y -16.094,A +3.800,E1 +0.105,E3 +5.131,E4 +5.131} C_DIS
 LIN_REL {X  +0.734,Y -23.794,A -0.997,E1 +1.118,E3 +7.793,E4 +7.793} C_DIS
 LIN_REL {X  +1.027,Y -33.665,A +3.633,E1 +0.609,E3 +11.312,E4 +11.312} C_DIS
 LIN_REL {X  +0.745,Y -37.564,A +10.062,E1 -1.297,E3 +12.930,E4 +12.930} C_DIS
 LIN_REL {X  +0.160,Y -43.446,A +7.136,E1 -1.236,E3 +15.310,E4 +15.310} C_DIS
 LIN_REL {X  -0.643,Y -46.463,A +1.818,E1 -0.189,E3 +16.789,E4 +16.789} C_DIS
 LIN_REL {X  -1.397,Y -55.132,A +0.224,E1 +0.346,E3 +20.701,E4 +20.701} C_DIS
 LIN_REL {X  -0.702,Y -73.363,A +0.634,E1 +0.296,E3 +30.090,E4 +30.090} C_DIS
 LIN_REL {X  +0.059,Y -225.709,A +0.001,E1 -0.020,E3 +95.671,E4 +95.671} C_DIS
 LIN_REL {X  +0.018,Y -43.522,A +0.000,E1 -0.003,E3 +18.467,E4 +18.467} C_DIS
 LIN_REL {X  +0.166,Y -31.307,A +0.000,E1 -0.018,E3 +13.420,E4 +13.420} C_DIS
 LIN_REL {X  +0.233,Y -13.270,A +0.000,E1 -0.022,E3 +5.816,E4 +5.816} C_DIS
 LIN_REL {X  +1.366,Y -27.298,A +0.000,E1 -0.126,E3 +12.650,E4 +12.650} C_DIS
 LIN_REL {X  +8.345,Y -41.089,A +0.000,E1 -0.766,E3 +23.837,E4 +23.837} C_DIS
 LIN_REL {X  +18.238,Y -32.330,A +0.001,E1 -1.935,E3 +25.376,E4 +25.376} C_DIS
 LIN_REL {X  +16.000,Y -14.360,A +3.516,E1 -1.834,E3 +12.887,E4 +12.887} C_DIS
 LIN_REL {X  +20.312,Y -16.924,A +11.171,E1 -4.697,E3 +20.568,E4 +20.568} C_DIS
 LIN_REL {X  +15.821,Y -22.718,A +7.098,E1 -4.956,E3 +32.172,E4 +32.172} C_DIS
 LIN_REL {X  +9.421,Y -23.866,A +6.736,E1 -4.437,E3 +41.036,E4 +41.036} C_DIS
 LIN_REL {X  +3.661,Y -25.092,A +1.450,E1 -5.412,E3 +53.988,E4 +53.988} C_DIS
 LIN_REL {X  -4.168,Y -20.869,A +0.028,E1 -6.472,E3 +62.125,E4 +62.125} C_DIS
 LIN_REL {X  -4.316,Y -2.000,A +0.000,E1 -4.216,E3 +33.264,E4 +33.264} C_DIS
 LIN_REL {X  -2.896,Y +12.706,A +0.000,E1 -6.125,E3 +31.047,E4 +31.047} C_DIS
 LIN_REL {X  -0.407,Y +27.885,A +0.000,E1 -13.058,E3 +26.838,E4 +26.838} C_DIS
 LIN_REL {X  -0.310,Y +28.969,A +0.000,E1 -18.562,E3 +20.747,E4 +20.747} C_DIS
 LIN_REL {X  -5.489,Y +18.847,A +0.000,E1 -18.099,E3 +17.557,E4 +17.557} C_DIS
 LIN_REL {X  -15.670,Y +12.857,A +0.000,E1 -17.750,E3 +20.222,E4 +20.222} C_DIS
 LIN_REL {X  -20.878,Y +15.155,A +0.000,E1 -18.026,E3 +16.880,E4 +16.880} C_DIS
 LIN_REL {X  -16.297,Y +16.840,A +0.000,E1 -9.740,E3 +11.900,E4 +11.900} C_DIS
ENDFOR

HALT
LIN {X -167.264,Y 528.355,Z 0.000,A 30.000, B 0.00, C 0.00,E1 -65.711}
HALT

; PLY 9 OF 41 (Connector)

; ANGLE 51.0 (Not valid for Circ layers and non-tubes)
$APO.CDIS=85
$VEL_EXTAX[1]=100
FOR N_CYC=1 to 1
 LIN_REL {X  +0.000,Y +6.378,A +0.000,E1 -1.210,E3 +1.854,E4 +1.854} C_DIS
 LIN_REL {X  +0.000,Y +14.621,A +0.000,E1 -2.616,E3 +4.458,E4 +4.458} C_DIS
 LIN_REL {X  +0.000,Y +32.005,A +0.000,E1 -3.259,E3 +10.675,E4 +10.675} C_DIS
 LIN_REL {X  +0.000,Y +40.708,A +0.000,E1 -1.459,E3 +13.747,E4 +13.747} C_DIS
 LIN_REL {X  +0.000,Y +26.153,A -0.784,E1 -0.105,E3 +9.652,E4 +9.652} C_DIS
 LIN_REL {X  +0.000,Y +20.741,A -5.442,E1 +0.518,E3 +8.145,E4 +8.145} C_DIS
 LIN_REL {X  +0.000,Y +25.002,A -2.452,E1 -0.784,E3 +10.228,E4 +10.228} C_DIS
 LIN_REL {X  +0.000,Y +35.423,A -8.939,E1 +0.931,E3 +14.590,E4 +14.590} C_DIS
 LIN_REL {X  +0.000,Y +43.889,A -6.529,E1 +0.797,E3 +18.871,E4 +18.871} C_DIS
 LIN_REL {X  +0.000,Y +59.890,A -4.616,E1 +0.603,E3 +29.034,E4 +29.034} C_DIS
 LIN_REL {X  +0.000,Y +47.666,A -1.237,E1 +1.513,E3 +37.044,E4 +37.044} C_DIS
 LIN_REL {X  +0.000,Y +43.953,A -0.001,E1 +3.475,E3 +52.262,E4 +52.262} C_DIS
 LIN_REL {X  +0.000,Y +54.086,A +0.000,E1 +3.862,E3 +65.301,E4 +65.301} C_DIS
 LIN_REL {X  +0.000,Y +63.043,A -0.000,E1 +4.449,E3 +82.404,E4 +82.404} C_DIS
 LIN_REL {X  +0.000,Y +67.569,A +0.000,E1 +5.026,E3 +100.105,E4 +100.105} C_DIS
 LIN_REL {X  +0.000,Y +60.598,A +0.000,E1 +4.978,E3 +104.421,E4 +104.421} C_DIS
 LIN_REL {X  +0.000,Y +45.881,A -0.000,E1 +4.244,E3 +91.905,E4 +91.905} C_DIS
 LIN_REL {X  +0.000,Y +33.669,A -0.000,E1 +3.512,E3 +77.261,E4 +77.261} C_DIS
 LIN_REL {X  +0.000,Y +23.775,A -0.000,E1 +3.184,E3 +61.446,E4 +61.446} C_DIS
 LIN_REL {X  +0.000,Y +13.031,A -0.000,E1 +2.930,E3 +36.561,E4 +36.561} C_DIS
 LIN_REL {X  +0.000,Y +8.579,A -0.001,E1 +1.393,E3 +26.568,E4 +26.568} C_DIS
 LIN_REL {X  +0.000,Y +15.457,A -0.005,E1 +1.280,E3 +46.740,E4 +46.740} C_DIS
 LIN_REL {X  +0.000,Y +16.398,A -0.038,E1 +2.723,E3 +57.821,E4 +57.821} C_DIS
 LIN_REL {X  +0.000,Y +11.283,A -0.160,E1 +1.949,E3 +43.088,E4 +43.088} C_DIS
 LIN_REL {X  +0.000,Y +7.051,A -0.286,E1 +0.917,E3 +27.945,E4 +27.945} C_DIS
 LIN_REL {X  +0.000,Y +6.762,A -0.405,E1 +1.621,E3 +30.217,E4 +30.217} C_DIS
 LIN_REL {X  +0.000,Y +7.005,A -1.131,E1 +1.696,E3 +28.761,E4 +28.761} C_DIS
 LIN_REL {X  +0.000,Y +7.141,A -7.654,E1 +6.428,E3 +31.676,E4 +31.676} C_DIS
 LIN_REL {X  +0.000,Y +3.401,A -14.382,E1 +15.617,E3 +29.067,E4 +29.067} C_DIS
 LIN_REL {X  +0.000,Y -0.692,A -5.741,E1 +9.583,E3 +24.085,E4 +24.085} C_DIS
 LIN_REL {X  +0.000,Y -6.981,A -0.197,E1 +8.163,E3 +40.575,E4 +40.575} C_DIS
 LIN_REL {X  +0.000,Y -7.790,A +0.000,E1 +6.568,E3 +35.728,E4 +35.728} C_DIS
 LIN_REL {X  +0.000,Y -3.628,A +0.000,E1 +1.649,E3 +14.520,E4 +14.520} C_DIS
ENDFOR

HALT
LIN {X -165.315,Y 1335.920,Z 0.000,A -29.910, B 0.00, C 0.00,E1 30.491}
HALT

; PLY 10 OF 41 (Helical)

; ANGLE 51.0 (Not valid for Circ layers and non-tubes)
$APO.CDIS=85
$VEL_EXTAX[1]=100
FOR N_CYC=1 to 21
 LIN_REL {X  +0.089,Y -11.136,A +1.567,E1 +3.050,E3 +26.385,E4 +26.385} C_DIS
 LIN_REL {X  +0.036,Y -9.284,A -1.129,E1 +2.814,E3 +20.702,E4 +20.702} C_DIS
 LIN_REL {X  +0.297,Y -8.859,A +6.194,E1 -0.666,E3 +19.682,E4 +19.682} C_DIS
 LIN_REL {X  +0.808,Y -13.517,A +13.981,E1 -4.951,E3 +32.712,E4 +32.712} C_DIS
 LIN_REL {X  +0.310,Y -9.680,A +6.467,E1 -3.232,E3 +26.549,E4 +26.549} C_DIS
 LIN_REL {X  -0.105,Y -12.353,A +2.141,E1 -0.721,E3 +37.803,E4 +37.803} C_DIS
 LIN_REL {X  +0.153,Y -14.590,A +0.505,E1 -0.125,E3 +48.668,E4 +48.668} C_DIS
 LIN_REL {X  -0.104,Y -19.134,A +0.164,E1 -0.475,E3 +66.192,E4 +66.192} C_DIS
 LIN_REL {X  +0.032,Y -26.591,A +0.019,E1 +0.112,E3 +91.145,E4 +91.145} C_DIS
 LIN_REL {X  +0.094,Y -551.955,A +0.001,E1 -0.007,E3 +1899.300,E4 +1899.300} C_DIS
 LIN_REL {X  -0.061,Y -28.620,A +0.002,E1 -0.035,E3 +98.592,E4 +98.592} C_DIS
 LIN_REL {X  +0.099,Y -20.079,A +0.000,E1 -0.077,E3 +69.371,E4 +69.371} C_DIS
 LIN_REL {X  +0.956,Y -15.336,A -0.005,E1 +0.010,E3 +52.823,E4 +52.823} C_DIS
 LIN_REL {X  +1.005,Y -9.310,A +0.015,E1 -0.057,E3 +33.219,E4 +33.219} C_DIS
 LIN_REL {X  +0.640,Y -6.016,A +0.061,E1 -0.256,E3 +22.163,E4 +22.163} C_DIS
 LIN_REL {X  +1.484,Y -10.990,A +0.831,E1 -0.886,E3 +41.508,E4 +41.508} C_DIS
 LIN_REL {X  +2.367,Y -8.825,A +7.631,E1 -7.546,E3 +45.384,E4 +45.384} C_DIS
 LIN_REL {X  +0.896,Y -3.315,A +13.716,E1 -15.686,E3 +41.139,E4 +41.139} C_DIS
 LIN_REL {X  -0.297,Y +0.786,A +7.140,E1 -10.329,E3 +25.702,E4 +25.702} C_DIS
 LIN_REL {X  -1.468,Y +5.522,A +0.521,E1 -7.898,E3 +41.124,E4 +41.124} C_DIS
 LIN_REL {X  -3.272,Y +15.142,A -0.131,E1 -10.512,E3 +53.162,E4 +53.162} C_DIS
 LIN_REL {X  -2.300,Y +12.529,A -2.905,E1 -3.815,E3 +31.734,E4 +31.734} C_DIS
 LIN_REL {X  -1.089,Y +10.506,A +1.524,E1 -3.960,E3 +24.140,E4 +24.140} C_DIS
 LIN_REL {X  -0.205,Y +8.815,A -3.304,E1 -0.712,E3 +19.761,E4 +19.761} C_DIS
 LIN_REL {X  +0.549,Y +13.054,A -11.060,E1 +2.722,E3 +30.762,E4 +30.762} C_DIS
 LIN_REL {X  +0.627,Y +17.255,A -10.666,E1 +4.694,E3 +46.980,E4 +46.980} C_DIS
 LIN_REL {X  -0.023,Y +15.398,A -3.237,E1 +1.325,E3 +48.568,E4 +48.568} C_DIS
 LIN_REL {X  +0.135,Y +17.872,A -0.132,E1 +0.618,E3 +61.054,E4 +61.054} C_DIS
 LIN_REL {X  -0.220,Y +23.475,A +0.002,E1 -0.166,E3 +80.707,E4 +80.707} C_DIS
 LIN_REL {X  +0.166,Y +33.220,A -0.002,E1 -0.019,E3 +114.254,E4 +114.254} C_DIS
 LIN_REL {X  +0.012,Y +531.310,A -0.001,E1 +0.004,E3 +1828.176,E4 +1828.176} C_DIS
 LIN_REL {X  -0.052,Y +28.617,A -0.001,E1 +0.036,E3 +98.584,E4 +98.584} C_DIS
 LIN_REL {X  +0.076,Y +20.104,A -0.011,E1 +0.079,E3 +69.426,E4 +69.426} C_DIS
 LIN_REL {X  +0.892,Y +15.381,A -0.041,E1 +0.014,E3 +52.948,E4 +52.948} C_DIS
 LIN_REL {X  +0.947,Y +9.327,A -0.077,E1 +0.101,E3 +33.264,E4 +33.264} C_DIS
 LIN_REL {X  +0.592,Y +6.005,A -0.136,E1 +0.316,E3 +22.105,E4 +22.105} C_DIS
 LIN_REL {X  +1.430,Y +10.966,A -0.500,E1 +0.636,E3 +41.041,E4 +41.041} C_DIS
 LIN_REL {X  +2.296,Y +8.175,A -3.798,E1 +4.053,E3 +39.816,E4 +39.816} C_DIS
 LIN_REL {X  +1.150,Y +3.631,A -11.276,E1 +11.580,E3 +31.219,E4 +31.219} C_DIS
 LIN_REL {X  -0.001,Y +0.510,A -11.397,E1 +13.305,E3 +25.652,E4 +25.652} C_DIS
 LIN_REL {X  -0.935,Y -1.511,A -2.754,E1 +7.102,E3 +26.931,E4 +26.931} C_DIS
 LIN_REL {X  -3.298,Y -5.564,A +0.745,E1 +6.649,E3 +40.343,E4 +40.343} C_DIS
 LIN_REL {X  -4.708,Y -20.935,A -0.664,E1 +12.911,E3 +58.258,E4 +58.258} C_DIS
ENDFOR

HALT
LIN {X -167.717,Y 1344.622,Z 0.000,A -18.303, B 0.00, C 0.00,E1 18.663}
HALT

; PLY 11 OF 41 (Connector)

; ANGLE 51.0 (Not valid for Circ layers and non-tubes)
$APO.CDIS=85
$VEL_EXTAX[1]=100
FOR N_CYC=1 to 1
 LIN_REL {X  +0.000,Y -6.749,A +0.974,E1 +3.425,E3 +21.375,E4 +21.375} C_DIS
 LIN_REL {X  +0.000,Y -11.547,A -2.399,E1 +4.958,E3 +34.836,E4 +34.836} C_DIS
 LIN_REL {X  +0.000,Y -12.185,A -6.347,E1 +7.536,E3 +24.576,E4 +24.576} C_DIS
 LIN_REL {X  +0.000,Y -10.217,A +1.978,E1 +1.903,E3 +18.633,E4 +18.633} C_DIS
 LIN_REL {X  +0.000,Y -12.984,A +11.637,E1 -3.135,E3 +26.047,E4 +26.047} C_DIS
 LIN_REL {X  +0.000,Y -10.179,A +7.669,E1 -2.821,E3 +22.921,E4 +22.921} C_DIS
 LIN_REL {X  +0.000,Y -15.543,A +3.623,E1 -0.270,E3 +35.593,E4 +35.593} C_DIS
 LIN_REL {X  +0.000,Y -23.700,A +0.864,E1 +1.824,E3 +51.728,E4 +51.728} C_DIS
 LIN_REL {X  +0.000,Y -30.611,A +0.251,E1 +2.486,E3 +61.789,E4 +61.789} C_DIS
 LIN_REL {X  +0.000,Y -39.306,A +0.049,E1 +3.161,E3 +71.713,E4 +71.713} C_DIS
 LIN_REL {X  +0.000,Y -53.537,A +0.004,E1 +3.972,E3 +86.184,E4 +86.184} C_DIS
 LIN_REL {X  +0.000,Y -64.573,A -0.000,E1 +4.213,E3 +90.064,E4 +90.064} C_DIS
 LIN_REL {X  +0.000,Y -70.724,A -0.000,E1 +4.042,E3 +84.993,E4 +84.993} C_DIS
 LIN_REL {X  +0.000,Y -78.542,A -0.000,E1 +3.959,E3 +81.114,E4 +81.114} C_DIS
 LIN_REL {X  +0.000,Y -83.435,A -0.000,E1 +3.728,E3 +73.654,E4 +73.654} C_DIS
 LIN_REL {X  +0.000,Y -85.371,A -0.000,E1 +3.407,E3 +64.167,E4 +64.167} C_DIS
 LIN_REL {X  +0.000,Y -91.935,A -0.000,E1 +3.287,E3 +58.326,E4 +58.326} C_DIS
 LIN_REL {X  +0.000,Y -95.986,A -0.000,E1 +3.072,E3 +50.600,E4 +50.600} C_DIS
 LIN_REL {X  +0.000,Y -97.035,A +0.001,E1 +2.772,E3 +41.893,E4 +41.893} C_DIS
 LIN_REL {X  +0.000,Y -80.674,A +0.025,E1 +2.107,E3 +29.313,E4 +29.313} C_DIS
 LIN_REL {X  +0.000,Y -59.470,A +0.980,E1 +1.132,E3 +25.037,E4 +25.037} C_DIS
 LIN_REL {X  +0.000,Y -45.258,A +3.624,E1 -0.067,E3 +27.732,E4 +27.732} C_DIS
 LIN_REL {X  +0.000,Y -32.162,A +7.778,E1 -1.250,E3 +28.270,E4 +28.270} C_DIS
 LIN_REL {X  +0.000,Y -20.839,A +11.240,E1 -3.274,E3 +26.885,E4 +26.885} C_DIS
 LIN_REL {X  +0.000,Y -15.818,A +5.990,E1 -6.619,E3 +32.257,E4 +32.257} C_DIS
 LIN_REL {X  +0.000,Y -3.510,A +0.360,E1 +1.377,E3 +14.035,E4 +14.035} C_DIS
 LIN_REL {X  +0.000,Y +4.557,A +0.002,E1 +6.548,E3 +8.652,E4 +8.652} C_DIS
 LIN_REL {X  +0.000,Y +11.890,A -0.000,E1 -2.836,E3 +15.274,E4 +15.274} C_DIS
 LIN_REL {X  +0.000,Y +32.887,A -0.000,E1 -11.086,E3 +35.585,E4 +35.585} C_DIS
 LIN_REL {X  +0.000,Y +47.616,A -0.000,E1 -9.199,E3 +34.604,E4 +34.604} C_DIS
 LIN_REL {X  +0.000,Y +32.625,A -0.000,E1 -8.789,E3 +17.179,E4 +17.179} C_DIS
 LIN_REL {X  +0.000,Y +20.055,A -0.000,E1 -18.285,E3 +8.659,E4 +8.659} C_DIS
 LIN_REL {X  +0.000,Y +0.575,A -0.000,E1 -3.117,E3 +0.575,E4 +0.575} C_DIS
 LIN_REL {X  +0.000,Y -8.107,A -0.000,E1 +20.949,E3 +0.184,E4 +0.184} C_DIS
 LIN_REL {X  +0.000,Y -5.814,A -0.000,E1 +12.353,E3 +0.111,E4 +0.111} C_DIS
 LIN_REL {X  +0.000,Y -8.338,A -0.000,E1 +1.513,E3 +0.111,E4 +0.111} C_DIS
 LIN_REL {X  +0.000,Y +3.105,A -0.000,E1 -8.242,E3 +0.147,E4 +0.147} C_DIS
 LIN_REL {X  +0.000,Y +17.593,A -0.000,E1 -6.458,E3 +4.518,E4 +4.518} C_DIS
 LIN_REL {X  +0.000,Y +29.681,A -0.000,E1 -12.959,E3 +11.481,E4 +11.481} C_DIS
 LIN_REL {X  +0.000,Y +32.488,A -0.000,E1 -20.228,E3 +11.406,E4 +11.406} C_DIS
 LIN_REL {X  +0.000,Y +25.632,A -0.000,E1 -18.878,E3 +8.199,E4 +8.199} C_DIS
 LIN_REL {X  +0.000,Y +26.743,A -0.000,E1 -18.556,E3 +7.969,E4 +7.969} C_DIS
 LIN_REL {X  +0.000,Y +27.333,A -0.000,E1 -14.173,E3 +8.381,E4 +8.381} C_DIS
 LIN_REL {X  +0.000,Y +24.634,A -0.000,E1 -9.794,E3 +6.910,E4 +6.910} C_DIS
 LIN_REL {X  +0.000,Y +13.462,A -0.000,E1 -3.768,E3 +3.755,E4 +3.755} C_DIS
 LIN_REL {X  +0.000,Y +10.872,A -0.000,E1 -2.572,E3 +2.944,E4 +2.944} C_DIS
 LIN_REL {X  +0.000,Y +14.337,A -0.000,E1 -2.945,E3 +3.665,E4 +3.665} C_DIS
 LIN_REL {X  +0.000,Y +23.039,A -0.000,E1 -3.317,E3 +6.107,E4 +6.107} C_DIS
 LIN_REL {X  +0.000,Y +36.664,A -0.000,E1 -3.158,E3 +10.016,E4 +10.016} C_DIS
 LIN_REL {X  +0.000,Y +15.660,A -0.000,E1 -0.509,E3 +4.994,E4 +4.994} C_DIS
 LIN_REL {X  +0.000,Y -5.380,A -0.000,E1 -0.467,E3 +1.274,E4 +1.274} C_DIS
 LIN_REL {X  +0.000,Y +21.577,A -0.911,E1 -0.752,E3 +6.932,E4 +6.932} C_DIS
 LIN_REL {X  +0.000,Y +28.710,A -8.086,E1 +0.422,E3 +9.791,E4 +9.791} C_DIS
 LIN_REL {X  +0.000,Y +18.045,A -4.972,E1 +1.360,E3 +6.319,E4 +6.319} C_DIS
 LIN_REL {X  +0.000,Y +16.319,A +2.388,E1 -1.467,E3 +5.785,E4 +5.785} C_DIS
 LIN_REL {X  +0.000,Y +17.890,A -1.841,E1 -0.710,E3 +6.565,E4 +6.565} C_DIS
 LIN_REL {X  +0.000,Y +32.212,A -7.227,E1 +0.996,E3 +12.141,E4 +12.141} C_DIS
 LIN_REL {X  +0.000,Y +47.871,A -5.087,E1 +0.597,E3 +18.710,E4 +18.710} C_DIS
 LIN_REL {X  +0.000,Y +68.722,A -3.501,E1 +0.198,E3 +28.777,E4 +28.777} C_DIS
 LIN_REL {X  +0.000,Y +89.832,A -0.762,E1 -0.145,E3 +41.583,E4 +41.583} C_DIS
 LIN_REL {X  +0.000,Y +302.093,A -0.001,E1 +0.005,E3 +141.913,E4 +141.913} C_DIS
 LIN_REL {X  +0.000,Y +257.345,A -0.002,E1 -0.000,E3 +120.872,E4 +120.872} C_DIS
 LIN_REL {X  +0.000,Y +66.803,A -0.301,E1 +0.023,E3 +31.483,E4 +31.483} C_DIS
 LIN_REL {X  +0.000,Y +47.705,A -2.050,E1 -0.300,E3 +24.755,E4 +24.755} C_DIS
 LIN_REL {X  +0.000,Y +41.854,A -7.267,E1 +0.318,E3 +30.220,E4 +30.220} C_DIS
 LIN_REL {X  +0.000,Y +28.430,A -13.013,E1 +3.082,E3 +30.428,E4 +30.428} C_DIS
 LIN_REL {X  +0.000,Y +14.893,A -6.784,E1 +3.146,E3 +22.284,E4 +22.284} C_DIS
 LIN_REL {X  +0.000,Y +15.160,A -0.583,E1 +5.813,E3 +35.188,E4 +35.188} C_DIS
 LIN_REL {X  +0.000,Y +4.905,A -0.000,E1 -1.357,E3 +16.288,E4 +16.288} C_DIS
 LIN_REL {X  +0.000,Y -4.218,A -0.000,E1 -6.614,E3 +7.202,E4 +7.202} C_DIS
 LIN_REL {X  +0.000,Y -12.176,A -0.000,E1 +0.422,E3 +11.080,E4 +11.080} C_DIS
 LIN_REL {X  +0.000,Y -28.307,A -0.000,E1 +9.223,E3 +25.870,E4 +25.870} C_DIS
 LIN_REL {X  +0.000,Y -46.487,A -0.000,E1 +11.292,E3 +33.734,E4 +33.734} C_DIS
 LIN_REL {X  +0.000,Y -33.211,A -0.000,E1 +6.717,E3 +18.604,E4 +18.604} C_DIS
 LIN_REL {X  +0.000,Y -23.967,A -0.000,E1 +11.188,E3 +11.028,E4 +11.028} C_DIS
 LIN_REL {X  +0.000,Y -9.965,A -0.000,E1 +13.923,E3 +4.393,E4 +4.393} C_DIS
 LIN_REL {X  +0.000,Y +7.934,A -0.000,E1 -21.033,E3 +0.027,E4 +0.027} C_DIS
 LIN_REL {X  +0.000,Y +5.752,A -0.000,E1 -12.400,E3 +0.016,E4 +0.016} C_DIS
 LIN_REL {X  +0.000,Y +8.223,A -0.000,E1 -1.504,E3 +0.017,E4 +0.017} C_DIS
 LIN_REL {X  +0.000,Y -3.465,A -0.000,E1 +8.346,E3 +0.022,E4 +0.022} C_DIS
 LIN_REL {X  +0.000,Y -17.890,A -0.000,E1 +6.566,E3 +4.250,E4 +4.250} C_DIS
 LIN_REL {X  +0.000,Y -29.989,A -0.000,E1 +13.137,E3 +10.933,E4 +10.933} C_DIS
 LIN_REL {X  +0.000,Y -32.710,A -0.000,E1 +20.352,E3 +10.796,E4 +10.796} C_DIS
 LIN_REL {X  +0.000,Y -25.733,A -0.000,E1 +18.812,E3 +7.697,E4 +7.697} C_DIS
 LIN_REL {X  +0.000,Y -26.880,A -0.000,E1 +18.392,E3 +7.380,E4 +7.380} C_DIS
 LIN_REL {X  +0.000,Y -28.065,A -0.000,E1 +14.330,E3 +7.643,E4 +7.643} C_DIS
 LIN_REL {X  +0.000,Y -29.079,A -0.000,E1 +10.853,E3 +7.247,E4 +7.247} C_DIS
ENDFOR

HALT
LIN {X -144.687,Y 1395.070,Z 0.000,A -30.000, B 0.00, C 0.00,E1 58.206}
HALT

; PLY 12 OF 41 (Helical)

; ANGLE 51.0 (Not valid for Circ layers and non-tubes)
$APO.CDIS=85
$VEL_EXTAX[1]=100
FOR N_CYC=1 to 56
 LIN_REL {X  -15.074,Y -29.767,A +0.000,E1 +9.092,E3 +14.973,E4 +14.973} C_DIS
 LIN_REL {X  -7.348,Y -47.000,A +0.000,E1 +5.660,E3 +14.939,E4 +14.939} C_DIS
 LIN_REL {X  -0.327,Y -30.116,A +0.043,E1 +1.483,E3 +10.093,E4 +10.093} C_DIS
 LIN_REL {X  +0.121,Y -22.217,A +4.925,E1 -0.225,E3 +7.540,E4 +7.540} C_DIS
 LIN_REL {X  +0.001,Y -14.273,A +7.593,E1 -0.769,E3 +4.894,E4 +4.894} C_DIS
 LIN_REL {X  -0.003,Y -13.874,A +1.451,E1 +0.056,E3 +4.815,E4 +4.815} C_DIS
 LIN_REL {X  +0.150,Y -18.128,A -3.628,E1 +1.179,E3 +6.456,E4 +6.456} C_DIS
 LIN_REL {X  +0.393,Y -19.754,A +1.762,E1 +0.363,E3 +7.298,E4 +7.298} C_DIS
 LIN_REL {X  +0.737,Y -36.562,A +7.200,E1 -0.410,E3 +14.048,E4 +14.048} C_DIS
 LIN_REL {X  +0.334,Y -54.526,A +7.100,E1 -0.905,E3 +21.857,E4 +21.857} C_DIS
 LIN_REL {X  -0.994,Y -70.820,A +3.004,E1 -0.164,E3 +30.138,E4 +30.138} C_DIS
 LIN_REL {X  -0.458,Y -89.648,A +0.549,E1 +0.288,E3 +41.804,E4 +41.804} C_DIS
 LIN_REL {X  +0.062,Y -235.310,A +0.001,E1 -0.021,E3 +112.139,E4 +112.139} C_DIS
 LIN_REL {X  +0.152,Y -74.946,A -0.000,E1 -0.019,E3 +35.853,E4 +35.853} C_DIS
 LIN_REL {X  +3.175,Y -60.274,A +0.000,E1 -0.317,E3 +31.142,E4 +31.142} C_DIS
 LIN_REL {X  +12.783,Y -42.940,A +0.000,E1 -1.342,E3 +29.777,E4 +29.777} C_DIS
 LIN_REL {X  +18.881,Y -23.861,A +0.460,E1 -2.257,E3 +21.845,E4 +21.845} C_DIS
 LIN_REL {X  +16.168,Y -12.681,A +8.201,E1 -2.958,E3 +14.090,E4 +14.090} C_DIS
 LIN_REL {X  +10.440,Y -8.657,A +8.183,E1 -2.988,E3 +12.321,E4 +12.321} C_DIS
 LIN_REL {X  +9.583,Y -9.951,A +1.367,E1 -1.482,E3 +16.338,E4 +16.338} C_DIS
 LIN_REL {X  +8.794,Y -10.954,A -2.966,E1 -0.519,E3 +21.888,E4 +21.888} C_DIS
 LIN_REL {X  +8.890,Y -13.825,A +4.159,E1 -4.536,E3 +35.358,E4 +35.358} C_DIS
 LIN_REL {X  +4.603,Y -12.186,A +9.243,E1 -10.006,E3 +40.370,E4 +40.370} C_DIS
 LIN_REL {X  -0.459,Y -9.939,A +1.353,E1 -8.668,E3 +41.144,E4 +41.144} C_DIS
 LIN_REL {X  -5.707,Y -9.687,A -0.000,E1 -7.235,E3 +52.061,E4 +52.061} C_DIS
 LIN_REL {X  -3.653,Y -1.626,A -0.000,E1 +0.440,E3 +20.599,E4 +20.599} C_DIS
 LIN_REL {X  -0.807,Y +8.764,A -0.000,E1 -4.910,E3 +17.201,E4 +17.201} C_DIS
 LIN_REL {X  -0.131,Y +24.325,A -0.000,E1 -15.273,E3 +25.891,E4 +25.891} C_DIS
 LIN_REL {X  -5.982,Y +24.543,A -0.000,E1 -21.681,E3 +28.284,E4 +28.284} C_DIS
 LIN_REL {X  -16.108,Y +12.581,A -0.000,E1 -18.650,E3 +25.038,E4 +25.038} C_DIS
 LIN_REL {X  -21.820,Y +15.911,A -0.000,E1 -19.262,E3 +21.987,E4 +21.987} C_DIS
 LIN_REL {X  -23.644,Y +28.209,A -0.000,E1 -14.788,E3 +19.735,E4 +19.735} C_DIS
 LIN_REL {X  -12.028,Y +35.197,A -0.000,E1 -7.539,E3 +13.489,E4 +13.489} C_DIS
 LIN_REL {X  -3.541,Y +41.796,A -0.000,E1 -3.288,E3 +12.972,E4 +12.972} C_DIS
 LIN_REL {X  +0.188,Y +26.499,A -0.196,E1 -1.297,E3 +9.096,E4 +9.096} C_DIS
 LIN_REL {X  +0.119,Y +17.359,A -5.827,E1 +0.391,E3 +5.950,E4 +5.950} C_DIS
 LIN_REL {X  +0.048,Y +16.741,A -9.460,E1 +0.994,E3 +5.812,E4 +5.812} C_DIS
 LIN_REL {X  +0.041,Y +12.774,A -1.992,E1 +0.090,E3 +4.494,E4 +4.494} C_DIS
 LIN_REL {X  +0.218,Y +22.174,A +5.187,E1 -1.444,E3 +7.992,E4 +7.992} C_DIS
 LIN_REL {X  +0.415,Y +23.026,A -1.173,E1 -0.516,E3 +8.595,E4 +8.595} C_DIS
 LIN_REL {X  +0.545,Y +32.843,A -6.810,E1 +0.806,E3 +12.687,E4 +12.687} C_DIS
 LIN_REL {X  +0.166,Y +50.909,A -5.567,E1 +0.644,E3 +20.490,E4 +20.490} C_DIS
 LIN_REL {X  -0.942,Y +71.381,A -3.781,E1 +0.185,E3 +30.556,E4 +30.556} C_DIS
 LIN_REL {X  -0.450,Y +84.555,A -0.380,E1 -0.263,E3 +39.493,E4 +39.493} C_DIS
 LIN_REL {X  +0.064,Y +235.368,A -0.001,E1 +0.022,E3 +112.097,E4 +112.097} C_DIS
 LIN_REL {X  +0.154,Y +75.707,A -0.000,E1 +0.019,E3 +36.194,E4 +36.194} C_DIS
 LIN_REL {X  +3.107,Y +59.558,A -0.000,E1 +0.317,E3 +30.788,E4 +30.788} C_DIS
 LIN_REL {X  +12.730,Y +42.891,A -0.000,E1 +1.344,E3 +29.752,E4 +29.752} C_DIS
 LIN_REL {X  +18.486,Y +23.738,A -0.375,E1 +2.222,E3 +21.647,E4 +21.647} C_DIS
 LIN_REL {X  +15.762,Y +12.225,A -7.129,E1 +2.795,E3 +13.517,E4 +13.517} C_DIS
 LIN_REL {X  +10.357,Y +7.718,A -9.304,E1 +3.163,E3 +11.327,E4 +11.327} C_DIS
 LIN_REL {X  +9.761,Y +9.024,A -3.219,E1 +2.078,E3 +15.204,E4 +15.204} C_DIS
 LIN_REL {X  +8.581,Y +10.150,A +2.726,E1 +0.536,E3 +19.865,E4 +19.865} C_DIS
 LIN_REL {X  +7.468,Y +11.001,A -3.485,E1 +3.399,E3 +26.323,E4 +26.323} C_DIS
 LIN_REL {X  +6.717,Y +15.381,A -7.240,E1 +9.456,E3 +46.684,E4 +46.684} C_DIS
 LIN_REL {X  +0.229,Y +13.738,A -1.973,E1 +9.620,E3 +52.944,E4 +52.944} C_DIS
 LIN_REL {X  -6.234,Y +9.630,A -0.001,E1 +7.184,E3 +49.634,E4 +49.634} C_DIS
 LIN_REL {X  -3.484,Y +1.205,A -0.000,E1 -0.288,E3 +19.054,E4 +19.054} C_DIS
 LIN_REL {X  -0.792,Y -9.029,A -0.000,E1 +4.952,E3 +17.037,E4 +17.037} C_DIS
 LIN_REL {X  -0.131,Y -24.443,A -0.000,E1 +15.273,E3 +25.906,E4 +25.906} C_DIS
 LIN_REL {X  -5.982,Y -24.632,A -0.000,E1 +21.680,E3 +28.283,E4 +28.283} C_DIS
 LIN_REL {X  -16.103,Y -12.651,A -0.000,E1 +18.647,E3 +25.033,E4 +25.033} C_DIS
 LIN_REL {X  -20.424,Y -14.811,A -0.000,E1 +18.261,E3 +20.576,E4 +20.576} C_DIS
 LIN_REL {X  -17.797,Y -17.833,A -0.000,E1 +11.381,E3 +13.879,E4 +13.879} C_DIS
ENDFOR

HALT
LIN {X -168.159,Y 1395.019,Z 0.000,A -30.000, B 0.00, C 0.00,E1 62.680}
HALT

; PLY 13 OF 41 (Connector)

; ANGLE 51.0 (Not valid for Circ layers and non-tubes)
$APO.CDIS=85
$VEL_EXTAX[1]=100
FOR N_CYC=1 to 1
 LIN_REL {X  +0.000,Y -9.931,A +0.000,E1 +2.034,E3 +3.713,E4 +3.713} C_DIS
 LIN_REL {X  +0.000,Y -15.219,A +0.000,E1 +2.603,E3 +6.116,E4 +6.116} C_DIS
 LIN_REL {X  +0.000,Y -28.602,A +0.000,E1 +3.185,E3 +11.353,E4 +11.353} C_DIS
 LIN_REL {X  +0.000,Y -32.667,A +0.000,E1 +1.759,E3 +11.751,E4 +11.751} C_DIS
 LIN_REL {X  +0.000,Y -4.269,A +0.000,E1 +0.040,E3 +3.684,E4 +3.684} C_DIS
 LIN_REL {X  +0.000,Y -11.353,A +0.002,E1 +0.574,E3 +5.370,E4 +5.370} C_DIS
 LIN_REL {X  +0.000,Y -30.702,A +1.667,E1 -0.263,E3 +11.897,E4 +11.897} C_DIS
 LIN_REL {X  +0.000,Y -21.345,A +8.058,E1 -0.871,E3 +8.807,E4 +8.807} C_DIS
 LIN_REL {X  +0.000,Y -12.398,A +1.018,E1 +0.751,E3 +5.946,E4 +5.946} C_DIS
 LIN_REL {X  +0.000,Y -19.430,A +1.002,E1 +0.019,E3 +9.238,E4 +9.238} C_DIS
 LIN_REL {X  +0.000,Y -35.290,A +6.056,E1 -0.755,E3 +16.617,E4 +16.617} C_DIS
 LIN_REL {X  +0.000,Y -52.427,A +7.945,E1 -0.996,E3 +26.931,E4 +26.931} C_DIS
 LIN_REL {X  +0.000,Y -52.006,A +4.002,E1 -1.210,E3 +37.415,E4 +37.415} C_DIS
 LIN_REL {X  +0.000,Y -52.888,A +0.249,E1 -2.773,E3 +52.831,E4 +52.831} C_DIS
 LIN_REL {X  +0.000,Y -60.838,A +0.001,E1 -3.115,E3 +65.149,E4 +65.149} C_DIS
 LIN_REL {X  +0.000,Y -69.223,A -0.000,E1 -3.580,E3 +80.716,E4 +80.716} C_DIS
 LIN_REL {X  +0.000,Y -73.314,A -0.000,E1 -3.968,E3 +95.333,E4 +95.333} C_DIS
 LIN_REL {X  +0.000,Y -66.651,A +0.000,E1 -3.882,E3 +97.918,E4 +97.918} C_DIS
 LIN_REL {X  +0.000,Y -63.587,A +0.000,E1 -4.068,E3 +106.239,E4 +106.239} C_DIS
 LIN_REL {X  +0.000,Y -54.705,A +0.000,E1 -3.914,E3 +104.399,E4 +104.399} C_DIS
 LIN_REL {X  +0.000,Y -41.720,A +0.005,E1 -3.566,E3 +90.377,E4 +90.377} C_DIS
 LIN_REL {X  +0.000,Y -27.945,A +0.157,E1 -2.997,E3 +66.491,E4 +66.491} C_DIS
 LIN_REL {X  +0.000,Y -19.510,A +1.581,E1 -1.872,E3 +47.111,E4 +47.111} C_DIS
 LIN_REL {X  +0.000,Y -13.314,A +7.900,E1 -6.014,E3 +35.958,E4 +35.958} C_DIS
 LIN_REL {X  +0.000,Y -6.208,A +12.793,E1 -13.799,E3 +26.060,E4 +26.060} C_DIS
 LIN_REL {X  +0.000,Y -1.824,A +5.470,E1 -7.527,E3 +12.771,E4 +12.771} C_DIS
 LIN_REL {X  +0.000,Y -1.175,A -2.198,E1 +0.663,E3 +12.539,E4 +12.539} C_DIS
 LIN_REL {X  +0.000,Y -0.621,A -3.128,E1 +1.647,E3 +14.007,E4 +14.007} C_DIS
 LIN_REL {X  +0.000,Y +1.132,A +4.499,E1 -8.454,E3 +17.695,E4 +17.695} C_DIS
 LIN_REL {X  +0.000,Y +6.204,A +2.893,E1 -10.749,E3 +26.326,E4 +26.326} C_DIS
 LIN_REL {X  +0.000,Y +24.036,A +0.028,E1 -16.376,E3 +43.956,E4 +43.956} C_DIS
ENDFOR

HALT
LIN {X -163.861,Y 569.550,Z 0.000,A 30.000, B 0.00, C 0.00,E1 -33.498}
HALT

; PLY 14 OF 41 (Helical)

; ANGLE 51.0 (Not valid for Circ layers and non-tubes)
$APO.CDIS=85
$VEL_EXTAX[1]=100
FOR N_CYC=1 to 30
 LIN_REL {X  -1.790,Y +19.836,A -0.123,E1 -7.165,E3 +25.508,E4 +25.508} C_DIS
 LIN_REL {X  -0.772,Y +12.435,A -4.676,E1 -0.852,E3 +16.408,E4 +16.408} C_DIS
 LIN_REL {X  -0.532,Y +8.678,A -6.964,E1 +1.472,E3 +12.093,E4 +12.093} C_DIS
 LIN_REL {X  -0.520,Y +9.312,A -1.210,E1 -0.861,E3 +13.708,E4 +13.708} C_DIS
 LIN_REL {X  -0.113,Y +7.583,A +4.664,E1 -3.054,E3 +11.664,E4 +11.664} C_DIS
 LIN_REL {X  +0.390,Y +8.503,A -2.022,E1 -0.577,E3 +13.521,E4 +13.521} C_DIS
 LIN_REL {X  +1.242,Y +16.633,A -10.842,E1 +2.843,E3 +28.336,E4 +28.336} C_DIS
 LIN_REL {X  +1.973,Y +24.399,A -7.365,E1 +2.164,E3 +45.844,E4 +45.844} C_DIS
 LIN_REL {X  +3.267,Y +34.969,A -1.413,E1 -0.715,E3 +70.269,E4 +70.269} C_DIS
 LIN_REL {X  +2.808,Y +38.562,A -0.048,E1 -0.565,E3 +80.055,E4 +80.055} C_DIS
 LIN_REL {X  +1.407,Y +44.698,A -0.001,E1 -0.021,E3 +94.414,E4 +94.414} C_DIS
 LIN_REL {X  +0.325,Y +52.589,A +0.000,E1 +0.036,E3 +111.815,E4 +111.815} C_DIS
 LIN_REL {X  +0.020,Y +338.406,A -0.000,E1 +0.004,E3 +720.250,E4 +720.250} C_DIS
 LIN_REL {X  -0.112,Y +52.679,A -0.000,E1 +0.027,E3 +112.219,E4 +112.219} C_DIS
 LIN_REL {X  -0.874,Y +48.890,A -0.001,E1 +0.319,E3 +104.871,E4 +104.871} C_DIS
 LIN_REL {X  -1.682,Y +39.667,A -0.020,E1 +1.224,E3 +87.309,E4 +87.309} C_DIS
 LIN_REL {X  +0.178,Y +27.430,A -0.233,E1 +1.921,E3 +64.024,E4 +64.024} C_DIS
 LIN_REL {X  +2.985,Y +16.504,A -1.555,E1 +2.288,E3 +42.783,E4 +42.783} C_DIS
 LIN_REL {X  +3.376,Y +9.383,A -7.522,E1 +6.088,E3 +29.993,E4 +29.993} C_DIS
 LIN_REL {X  +2.384,Y +5.772,A -12.981,E1 +11.640,E3 +25.467,E4 +25.467} C_DIS
 LIN_REL {X  +0.878,Y +2.094,A -4.086,E1 +4.921,E3 +13.171,E4 +13.171} C_DIS
 LIN_REL {X  +1.068,Y +1.669,A +4.166,E1 -1.030,E3 +18.301,E4 +18.301} C_DIS
 LIN_REL {X  +0.779,Y +0.217,A -0.159,E1 +3.275,E3 +19.724,E4 +19.724} C_DIS
 LIN_REL {X  -0.248,Y -1.574,A -5.556,E1 +9.118,E3 +18.830,E4 +18.830} C_DIS
 LIN_REL {X  -3.385,Y -7.281,A -2.053,E1 +12.352,E3 +36.332,E4 +36.332} C_DIS
 LIN_REL {X  -8.943,Y -21.008,A +0.000,E1 +16.823,E3 +49.511,E4 +49.511} C_DIS
 LIN_REL {X  -4.828,Y -22.813,A +0.003,E1 +10.277,E3 +33.331,E4 +33.331} C_DIS
 LIN_REL {X  -1.574,Y -16.042,A +3.360,E1 +2.890,E3 +21.228,E4 +21.228} C_DIS
 LIN_REL {X  -0.854,Y -11.706,A +7.814,E1 -1.173,E3 +16.151,E4 +16.151} C_DIS
 LIN_REL {X  -0.505,Y -8.930,A -0.323,E1 +1.497,E3 +13.022,E4 +13.022} C_DIS
 LIN_REL {X  -0.050,Y -7.488,A -4.382,E1 +2.896,E3 +11.327,E4 +11.327} C_DIS
 LIN_REL {X  +0.453,Y -8.819,A +2.986,E1 +0.290,E3 +13.827,E4 +13.827} C_DIS
 LIN_REL {X  +1.096,Y -15.174,A +11.720,E1 -3.278,E3 +25.548,E4 +25.548} C_DIS
 LIN_REL {X  +1.095,Y -15.246,A +6.268,E1 -2.116,E3 +27.975,E4 +27.975} C_DIS
 LIN_REL {X  +2.017,Y -23.729,A +2.102,E1 +0.164,E3 +46.465,E4 +46.465} C_DIS
 LIN_REL {X  +3.054,Y -32.661,A +0.403,E1 +0.885,E3 +66.539,E4 +66.539} C_DIS
 LIN_REL {X  +2.391,Y -37.907,A +0.047,E1 +0.334,E3 +79.107,E4 +79.107} C_DIS
 LIN_REL {X  +1.075,Y -44.605,A +0.002,E1 -0.024,E3 +94.391,E4 +94.391} C_DIS
 LIN_REL {X  +0.217,Y -52.691,A -0.000,E1 -0.027,E3 +112.032,E4 +112.032} C_DIS
 LIN_REL {X  +0.009,Y -328.940,A +0.000,E1 -0.003,E3 +699.830,E4 +699.830} C_DIS
 LIN_REL {X  -0.114,Y -52.701,A +0.000,E1 -0.025,E3 +112.222,E4 +112.222} C_DIS
 LIN_REL {X  -0.879,Y -48.904,A +0.000,E1 -0.321,E3 +104.859,E4 +104.859} C_DIS
 LIN_REL {X  -1.647,Y -39.676,A +0.005,E1 -1.214,E3 +87.302,E4 +87.302} C_DIS
 LIN_REL {X  +0.171,Y -27.606,A +0.218,E1 -1.883,E3 +64.372,E4 +64.372} C_DIS
 LIN_REL {X  +2.867,Y -16.673,A +2.403,E1 -2.811,E3 +43.339,E4 +43.339} C_DIS
 LIN_REL {X  +3.676,Y -10.511,A +9.757,E1 -8.096,E3 +34.611,E4 +34.611} C_DIS
 LIN_REL {X  +2.107,Y -5.098,A +10.509,E1 -10.104,E3 +23.898,E4 +23.898} C_DIS
 LIN_REL {X  +0.883,Y -1.805,A +0.918,E1 -2.238,E3 +12.418,E4 +12.418} C_DIS
 LIN_REL {X  +1.262,Y -1.463,A -4.827,E1 +1.655,E3 +18.826,E4 +18.826} C_DIS
 LIN_REL {X  +0.600,Y +0.010,A +2.445,E1 -4.639,E3 +15.641,E4 +15.641} C_DIS
 LIN_REL {X  -0.702,Y +2.279,A +7.727,E1 -12.857,E3 +25.877,E4 +25.877} C_DIS
 LIN_REL {X  -4.256,Y +6.826,A +0.845,E1 -10.896,E3 +33.044,E4 +33.044} C_DIS
 LIN_REL {X  -11.673,Y +31.028,A +0.000,E1 -20.858,E3 +63.065,E4 +63.065} C_DIS
ENDFOR

HALT
LIN {X -168.596,Y 567.662,Z 0.000,A 30.000, B 0.00, C 0.00,E1 -33.996}
HALT

; PLY 15 OF 41 (Connector)

; ANGLE 51.0 (Not valid for Circ layers and non-tubes)
$APO.CDIS=85
$VEL_EXTAX[1]=100
FOR N_CYC=1 to 1
 LIN_REL {X  +0.000,Y +13.174,A +0.000,E1 -4.073,E3 +16.637,E4 +16.637} C_DIS
 LIN_REL {X  +0.000,Y +21.225,A -2.211,E1 -4.895,E3 +24.628,E4 +24.628} C_DIS
 LIN_REL {X  +0.000,Y +12.570,A -7.532,E1 +1.015,E3 +16.424,E4 +16.424} C_DIS
 LIN_REL {X  +0.000,Y +10.495,A -0.532,E1 -1.394,E3 +14.186,E4 +14.186} C_DIS
 LIN_REL {X  +0.000,Y +11.190,A -1.570,E1 -1.428,E3 +14.392,E4 +14.392} C_DIS
 LIN_REL {X  +0.000,Y +18.046,A -10.752,E1 +2.241,E3 +25.282,E4 +25.282} C_DIS
 LIN_REL {X  +0.000,Y +19.354,A -5.644,E1 +0.921,E3 +29.058,E4 +29.058} C_DIS
 LIN_REL {X  +0.000,Y +29.061,A -1.559,E1 -1.182,E3 +43.676,E4 +43.676} C_DIS
 LIN_REL {X  +0.000,Y +37.695,A -0.188,E1 -1.826,E3 +54.238,E4 +54.238} C_DIS
 LIN_REL {X  +0.000,Y +49.185,A -0.011,E1 -2.401,E3 +65.673,E4 +65.673} C_DIS
 LIN_REL {X  +0.000,Y +61.291,A -0.001,E1 -2.859,E3 +74.334,E4 +74.334} C_DIS
 LIN_REL {X  +0.000,Y +75.615,A +0.000,E1 -3.227,E3 +81.759,E4 +81.759} C_DIS
 LIN_REL {X  +0.000,Y +79.850,A +0.000,E1 -3.094,E3 +76.200,E4 +76.200} C_DIS
 LIN_REL {X  +0.000,Y +84.499,A +0.000,E1 -2.984,E3 +70.876,E4 +70.876} C_DIS
 LIN_REL {X  +0.000,Y +86.084,A -0.000,E1 -2.782,E3 +63.215,E4 +63.215} C_DIS
 LIN_REL {X  +0.000,Y +91.876,A -0.000,E1 -2.722,E3 +58.643,E4 +58.643} C_DIS
 LIN_REL {X  +0.000,Y +94.840,A -0.000,E1 -2.575,E3 +52.031,E4 +52.031} C_DIS
 LIN_REL {X  +0.000,Y +94.364,A -0.011,E1 -2.343,E3 +44.135,E4 +44.135} C_DIS
 LIN_REL {X  +0.000,Y +76.880,A -0.228,E1 -1.727,E3 +31.472,E4 +31.472} C_DIS
 LIN_REL {X  +0.000,Y +58.753,A -2.075,E1 -0.869,E3 +27.469,E4 +27.469} C_DIS
 LIN_REL {X  +0.000,Y +44.133,A -7.388,E1 +0.691,E3 +30.636,E4 +30.636} C_DIS
 LIN_REL {X  +0.000,Y +32.532,A -12.832,E1 +3.688,E3 +31.442,E4 +31.442} C_DIS
 LIN_REL {X  +0.000,Y +19.241,A -6.728,E1 +4.112,E3 +27.143,E4 +27.143} C_DIS
 LIN_REL {X  +0.000,Y +11.793,A -0.738,E1 +2.724,E3 +30.067,E4 +30.067} C_DIS
 LIN_REL {X  +0.000,Y -2.853,A +0.000,E1 -1.749,E3 +20.954,E4 +20.954} C_DIS
 LIN_REL {X  +0.000,Y -17.834,A +0.000,E1 +2.242,E3 +24.136,E4 +24.136} C_DIS
 LIN_REL {X  +0.000,Y -39.640,A +0.000,E1 +10.817,E3 +35.542,E4 +35.542} C_DIS
 LIN_REL {X  +0.000,Y -25.822,A +0.000,E1 +7.968,E3 +17.738,E4 +17.738} C_DIS
 LIN_REL {X  +0.000,Y -1.533,A +0.000,E1 -0.268,E3 +1.207,E4 +1.207} C_DIS
 LIN_REL {X  +0.000,Y +8.963,A +0.000,E1 -10.218,E3 +0.740,E4 +0.740} C_DIS
 LIN_REL {X  +0.000,Y -1.888,A +0.000,E1 -2.329,E3 +0.537,E4 +0.537} C_DIS
 LIN_REL {X  +0.000,Y -16.977,A +0.000,E1 +8.911,E3 +6.910,E4 +6.910} C_DIS
 LIN_REL {X  +0.000,Y -42.216,A +0.000,E1 +17.221,E3 +19.332,E4 +19.332} C_DIS
 LIN_REL {X  +0.000,Y -37.774,A +0.000,E1 +19.595,E3 +14.105,E4 +14.105} C_DIS
 LIN_REL {X  +0.000,Y -18.395,A +0.000,E1 +19.599,E3 +5.763,E4 +5.763} C_DIS
 LIN_REL {X  +0.000,Y -4.113,A +0.000,E1 +5.797,E3 +1.159,E4 +1.159} C_DIS
 LIN_REL {X  +0.000,Y +5.056,A +0.000,E1 -21.240,E3 +0.132,E4 +0.132} C_DIS
 LIN_REL {X  +0.000,Y +6.411,A +0.000,E1 -9.204,E3 +0.105,E4 +0.105} C_DIS
 LIN_REL {X  +0.000,Y -4.206,A +0.000,E1 +12.792,E3 +0.132,E4 +0.132} C_DIS
 LIN_REL {X  +0.000,Y -23.115,A +0.000,E1 +16.873,E3 +7.950,E4 +7.950} C_DIS
 LIN_REL {X  +0.000,Y -28.702,A +0.000,E1 +18.449,E3 +9.079,E4 +9.079} C_DIS
 LIN_REL {X  +0.000,Y -46.232,A +0.000,E1 +20.816,E3 +16.539,E4 +16.539} C_DIS
ENDFOR

HALT
LIN {X -147.860,Y 1392.241,Z 0.000,A -30.000, B 0.00, C 0.00,E1 56.905}
HALT

; PLY 16 OF 41 (Helical)

; ANGLE 51.0 (Not valid for Circ layers and non-tubes)
$APO.CDIS=85
$VEL_EXTAX[1]=100
FOR N_CYC=1 to 56
 LIN_REL {X  -14.867,Y -35.476,A +0.000,E1 +9.823,E3 +19.147,E4 +19.147} C_DIS
 LIN_REL {X  -5.107,Y -40.909,A +0.000,E1 +4.652,E3 +14.380,E4 +14.380} C_DIS
 LIN_REL {X  -0.584,Y -22.630,A +0.207,E1 +0.815,E3 +7.708,E4 +7.708} C_DIS
 LIN_REL {X  -0.018,Y -13.983,A +0.347,E1 +0.645,E3 +5.131,E4 +5.131} C_DIS
 LIN_REL {X  +0.063,Y -19.835,A +7.368,E1 -0.405,E3 +7.564,E4 +7.564} C_DIS
 LIN_REL {X  +0.011,Y -21.382,A +3.887,E1 -0.117,E3 +8.343,E4 +8.343} C_DIS
 LIN_REL {X  +0.268,Y -23.831,A -0.549,E1 +0.762,E3 +9.625,E4 +9.625} C_DIS
 LIN_REL {X  +0.673,Y -32.878,A +5.677,E1 +0.003,E3 +13.872,E4 +13.872} C_DIS
 LIN_REL {X  +0.492,Y -48.483,A +7.882,E1 -0.812,E3 +21.412,E4 +21.412} C_DIS
 LIN_REL {X  -0.636,Y -66.677,A +4.438,E1 -0.394,E3 +31.379,E4 +31.379} C_DIS
 LIN_REL {X  -0.378,Y -81.951,A +0.732,E1 +0.271,E3 +42.097,E4 +42.097} C_DIS
 LIN_REL {X  +0.112,Y -265.682,A +0.011,E1 -0.027,E3 +139.723,E4 +139.723} C_DIS
 LIN_REL {X  +0.099,Y -71.712,A +0.000,E1 -0.014,E3 +37.809,E4 +37.809} C_DIS
 LIN_REL {X  +1.797,Y -56.391,A +0.000,E1 -0.214,E3 +31.116,E4 +31.116} C_DIS
 LIN_REL {X  +8.254,Y -43.602,A +0.000,E1 -0.938,E3 +29.249,E4 +29.249} C_DIS
 LIN_REL {X  +16.692,Y -29.890,A +0.046,E1 -2.123,E3 +26.508,E4 +26.508} C_DIS
 LIN_REL {X  +16.910,Y -15.467,A +5.547,E1 -2.849,E3 +16.712,E4 +16.712} C_DIS
 LIN_REL {X  +10.853,Y -8.042,A +8.333,E1 -3.007,E3 +11.686,E4 +11.686} C_DIS
 LIN_REL {X  +11.037,Y -8.779,A +3.318,E1 -2.463,E3 +15.583,E4 +15.583} C_DIS
 LIN_REL {X  +11.455,Y -14.401,A +4.074,E1 -4.379,E3 +28.571,E4 +28.571} C_DIS
 LIN_REL {X  +5.961,Y -11.618,A +6.931,E1 -5.129,E3 +25.975,E4 +25.975} C_DIS
 LIN_REL {X  +3.689,Y -13.311,A +1.698,E1 -5.394,E3 +33.383,E4 +33.383} C_DIS
 LIN_REL {X  -0.686,Y -17.703,A +0.053,E1 -6.585,E3 +52.380,E4 +52.380} C_DIS
 LIN_REL {X  -1.828,Y -0.654,A -0.000,E1 -2.875,E3 +33.458,E4 +33.458} C_DIS
 LIN_REL {X  +0.301,Y +12.220,A -0.000,E1 -9.985,E3 +30.125,E4 +30.125} C_DIS
 LIN_REL {X  -0.483,Y +13.767,A -0.000,E1 -11.754,E3 +22.302,E4 +22.302} C_DIS
 LIN_REL {X  -0.929,Y +12.998,A -0.000,E1 -5.910,E3 +18.319,E4 +18.319} C_DIS
 LIN_REL {X  -4.469,Y +9.738,A -0.000,E1 -10.697,E3 +18.333,E4 +18.333} C_DIS
 LIN_REL {X  -16.127,Y +12.706,A -0.000,E1 -19.779,E3 +31.195,E4 +31.195} C_DIS
 LIN_REL {X  -20.882,Y +15.217,A -0.000,E1 -19.668,E3 +26.426,E4 +26.426} C_DIS
 LIN_REL {X  -24.478,Y +28.146,A -0.000,E1 -17.323,E3 +25.236,E4 +25.236} C_DIS
 LIN_REL {X  -14.358,Y +40.828,A -0.000,E1 -9.504,E3 +18.690,E4 +18.690} C_DIS
 LIN_REL {X  -2.889,Y +33.493,A -0.003,E1 -3.060,E3 +11.510,E4 +11.510} C_DIS
 LIN_REL {X  -0.519,Y +32.349,A -0.161,E1 -1.349,E3 +11.374,E4 +11.374} C_DIS
 LIN_REL {X  +0.092,Y +17.745,A -6.168,E1 +0.264,E3 +6.755,E4 +6.755} C_DIS
 LIN_REL {X  +0.014,Y +18.501,A -6.676,E1 +0.428,E3 +7.181,E4 +7.181} C_DIS
 LIN_REL {X  +0.074,Y +25.655,A +0.382,E1 -0.497,E3 +10.224,E4 +10.224} C_DIS
 LIN_REL {X  +0.449,Y +27.610,A -2.332,E1 -0.435,E3 +11.487,E4 +11.487} C_DIS
 LIN_REL {X  +0.614,Y +40.448,A -6.860,E1 +0.474,E3 +17.579,E4 +17.579} C_DIS
 LIN_REL {X  -0.062,Y +59.403,A -6.092,E1 +0.694,E3 +27.270,E4 +27.270} C_DIS
 LIN_REL {X  -0.707,Y +76.212,A -2.046,E1 -0.149,E3 +38.056,E4 +38.056} C_DIS
 LIN_REL {X  +0.106,Y +87.706,A -0.044,E1 -0.030,E3 +45.938,E4 +45.938} C_DIS
 LIN_REL {X  +0.020,Y +205.666,A -0.000,E1 +0.008,E3 +108.030,E4 +108.030} C_DIS
 LIN_REL {X  +0.099,Y +75.436,A -0.000,E1 +0.014,E3 +39.709,E4 +39.709} C_DIS
 LIN_REL {X  +2.110,Y +60.133,A -0.000,E1 +0.247,E3 +33.273,E4 +33.273} C_DIS
 LIN_REL {X  +9.094,Y +42.645,A -0.000,E1 +1.034,E3 +29.281,E4 +29.281} C_DIS
 LIN_REL {X  +15.577,Y +27.201,A -0.061,E1 +1.997,E3 +24.262,E4 +24.262} C_DIS
 LIN_REL {X  +15.437,Y +14.417,A -3.772,E1 +2.336,E3 +15.164,E4 +15.164} C_DIS
 LIN_REL {X  +11.613,Y +8.613,A -9.614,E1 +3.312,E3 +12.102,E4 +12.102} C_DIS
 LIN_REL {X  +8.192,Y +6.112,A -4.970,E1 +2.334,E3 +10.760,E4 +10.760} C_DIS
 LIN_REL {X  +11.561,Y +12.346,A -2.283,E1 +3.049,E3 +23.399,E4 +23.399} C_DIS
 LIN_REL {X  +9.134,Y +16.800,A -6.868,E1 +6.232,E3 +35.627,E4 +35.627} C_DIS
 LIN_REL {X  +4.235,Y +18.651,A -2.409,E1 +7.477,E3 +46.561,E4 +46.561} C_DIS
 LIN_REL {X  -1.749,Y +14.204,A -0.023,E1 +5.139,E3 +45.885,E4 +45.885} C_DIS
 LIN_REL {X  -0.957,Y -3.344,A +0.000,E1 +4.505,E3 +35.944,E4 +35.944} C_DIS
 LIN_REL {X  +0.044,Y -17.055,A +0.000,E1 +14.555,E3 +34.357,E4 +34.357} C_DIS
 LIN_REL {X  -0.677,Y -13.170,A +0.000,E1 +9.067,E3 +19.187,E4 +19.187} C_DIS
 LIN_REL {X  -1.858,Y -11.368,A +0.000,E1 +6.416,E3 +17.079,E4 +17.079} C_DIS
 LIN_REL {X  -8.698,Y -10.680,A +0.000,E1 +14.460,E3 +23.713,E4 +23.713} C_DIS
 LIN_REL {X  -18.004,Y -12.556,A +0.000,E1 +19.256,E3 +28.555,E4 +28.555} C_DIS
 LIN_REL {X  -19.214,Y -15.661,A +0.000,E1 +16.740,E3 +20.019,E4 +20.019} C_DIS
 LIN_REL {X  -15.968,Y -17.845,A +0.000,E1 +10.856,E3 +16.996,E4 +16.996} C_DIS
ENDFOR

HALT
LIN {X -169.042,Y 1392.442,Z 0.000,A -30.000, B 0.00, C 0.00,E1 60.750}
HALT

; PLY 17 OF 41 (Connector)

; ANGLE 51.0 (Not valid for Circ layers and non-tubes)
$APO.CDIS=85
$VEL_EXTAX[1]=100
FOR N_CYC=1 to 1
 LIN_REL {X  +0.000,Y -10.439,A +0.000,E1 +1.856,E3 +6.041,E4 +6.041} C_DIS
 LIN_REL {X  +0.000,Y -25.509,A +0.000,E1 +4.046,E3 +14.194,E4 +14.194} C_DIS
 LIN_REL {X  +0.000,Y -22.722,A +0.000,E1 +2.302,E3 +9.459,E4 +9.459} C_DIS
 LIN_REL {X  +0.000,Y -4.328,A +0.000,E1 +0.456,E3 +3.672,E4 +3.672} C_DIS
 LIN_REL {X  +0.000,Y -26.264,A +0.000,E1 +1.107,E3 +8.977,E4 +8.977} C_DIS
 LIN_REL {X  +0.000,Y -12.176,A +0.004,E1 +0.401,E3 +6.640,E4 +6.640} C_DIS
 LIN_REL {X  +0.000,Y -19.844,A +0.987,E1 -0.066,E3 +9.000,E4 +9.000} C_DIS
 LIN_REL {X  +0.000,Y -21.380,A +6.812,E1 -0.660,E3 +9.832,E4 +9.832} C_DIS
 LIN_REL {X  +0.000,Y -12.774,A +3.059,E1 +0.042,E3 +6.518,E4 +6.518} C_DIS
 LIN_REL {X  +0.000,Y -24.637,A +2.011,E1 +0.165,E3 +12.883,E4 +12.883} C_DIS
 LIN_REL {X  +0.000,Y -38.624,A +6.737,E1 -0.745,E3 +20.623,E4 +20.623} C_DIS
 LIN_REL {X  +0.000,Y -51.215,A +7.947,E1 -1.197,E3 +31.396,E4 +31.396} C_DIS
 LIN_REL {X  +0.000,Y -54.569,A +2.352,E1 -1.351,E3 +43.871,E4 +43.871} C_DIS
 LIN_REL {X  +0.000,Y -60.291,A +0.090,E1 -1.717,E3 +53.454,E4 +53.454} C_DIS
 LIN_REL {X  +0.000,Y -71.987,A +0.001,E1 -2.026,E3 +67.983,E4 +67.983} C_DIS
 LIN_REL {X  +0.000,Y -78.670,A -0.000,E1 -2.268,E3 +79.830,E4 +79.830} C_DIS
 LIN_REL {X  +0.000,Y -76.919,A +0.000,E1 -2.299,E3 +84.361,E4 +84.361} C_DIS
 LIN_REL {X  +0.000,Y -74.797,A +0.000,E1 -2.334,E3 +88.765,E4 +88.765} C_DIS
 LIN_REL {X  +0.000,Y -72.372,A +0.000,E1 -2.378,E3 +93.042,E4 +93.042} C_DIS
 LIN_REL {X  +0.000,Y -59.526,A +0.004,E1 -2.133,E3 +82.507,E4 +82.507} C_DIS
 LIN_REL {X  +0.000,Y -42.278,A +0.162,E1 -1.804,E3 +62.171,E4 +62.171} C_DIS
 LIN_REL {X  +0.000,Y -29.208,A +1.771,E1 -1.231,E3 +43.799,E4 +43.799} C_DIS
 LIN_REL {X  +0.000,Y -21.202,A +8.761,E1 -4.965,E3 +36.205,E4 +36.205} C_DIS
 LIN_REL {X  +0.000,Y -11.495,A +13.705,E1 -12.632,E3 +27.500,E4 +27.500} C_DIS
 LIN_REL {X  +0.000,Y -4.953,A +4.525,E1 -6.131,E3 +18.203,E4 +18.203} C_DIS
 LIN_REL {X  +0.000,Y -1.768,A +1.058,E1 -6.956,E3 +31.122,E4 +31.122} C_DIS
 LIN_REL {X  +0.000,Y +9.094,A +0.014,E1 -13.049,E3 +40.916,E4 +40.916} C_DIS
 LIN_REL {X  +0.000,Y +21.402,A -0.000,E1 -15.430,E3 +34.759,E4 +34.759} C_DIS
 LIN_REL {X  +0.000,Y +22.950,A -0.000,E1 -13.807,E3 +22.376,E4 +22.376} C_DIS
 LIN_REL {X  +0.000,Y +14.002,A -0.000,E1 -6.816,E3 +11.708,E4 +11.708} C_DIS
ENDFOR

HALT
LIN {X -160.460,Y 552.324,Z 0.000,A 30.000, B 0.00, C 0.00,E1 -38.095}
HALT

; PLY 18 OF 41 (Helical)

; ANGLE 51.0 (Not valid for Circ layers and non-tubes)
$APO.CDIS=85
$VEL_EXTAX[1]=100
FOR N_CYC=1 to 41
 LIN_REL {X  -5.459,Y +28.114,A +0.000,E1 -9.986,E3 +26.382,E4 +26.382} C_DIS
 LIN_REL {X  -2.378,Y +28.454,A -0.022,E1 -4.822,E3 +24.890,E4 +24.890} C_DIS
 LIN_REL {X  -0.183,Y +15.295,A -3.544,E1 -0.580,E3 +14.267,E4 +14.267} C_DIS
 LIN_REL {X  -0.196,Y +15.833,A -7.076,E1 +0.771,E3 +15.566,E4 +15.566} C_DIS
 LIN_REL {X  -0.006,Y +11.111,A -0.091,E1 -0.944,E3 +11.487,E4 +11.487} C_DIS
 LIN_REL {X  +0.431,Y +13.498,A -3.757,E1 -0.050,E3 +14.719,E4 +14.719} C_DIS
 LIN_REL {X  +0.762,Y +23.526,A -9.952,E1 +2.087,E3 +27.446,E4 +27.446} C_DIS
 LIN_REL {X  +0.946,Y +38.203,A -5.078,E1 +0.804,E3 +48.613,E4 +48.613} C_DIS
 LIN_REL {X  +1.456,Y +46.351,A -0.467,E1 -0.327,E3 +61.956,E4 +61.956} C_DIS
 LIN_REL {X  +0.916,Y +54.342,A -0.013,E1 -0.014,E3 +73.825,E4 +73.825} C_DIS
 LIN_REL {X  +0.217,Y +71.553,A +0.000,E1 +0.036,E3 +97.780,E4 +97.780} C_DIS
 LIN_REL {X  +0.006,Y +316.774,A -0.000,E1 +0.005,E3 +433.271,E4 +433.271} C_DIS
 LIN_REL {X  -0.015,Y +37.312,A -0.000,E1 +0.018,E3 +51.076,E4 +51.076} C_DIS
 LIN_REL {X  +0.004,Y +28.280,A -0.000,E1 +0.074,E3 +38.847,E4 +38.847} C_DIS
 LIN_REL {X  +0.077,Y +16.611,A -0.000,E1 +0.112,E3 +22.991,E4 +22.991} C_DIS
 LIN_REL {X  +0.240,Y +15.534,A -0.002,E1 +0.196,E3 +21.759,E4 +21.759} C_DIS
 LIN_REL {X  +1.279,Y +26.262,A -0.012,E1 +0.665,E3 +37.899,E4 +37.899} C_DIS
 LIN_REL {X  +5.121,Y +31.582,A -0.182,E1 +1.757,E3 +49.378,E4 +49.378} C_DIS
 LIN_REL {X  +7.300,Y +18.011,A -1.679,E1 +2.192,E3 +32.385,E4 +32.385} C_DIS
 LIN_REL {X  +7.364,Y +10.957,A -8.101,E1 +5.176,E3 +24.891,E4 +24.891} C_DIS
 LIN_REL {X  +5.603,Y +6.788,A -10.479,E1 +7.421,E3 +21.021,E4 +21.021} C_DIS
 LIN_REL {X  +6.117,Y +5.814,A -4.820,E1 +6.646,E3 +29.521,E4 +29.521} C_DIS
 LIN_REL {X  +3.336,Y +2.616,A -4.641,E1 +8.630,E3 +27.469,E4 +27.469} C_DIS
 LIN_REL {X  -0.267,Y -0.366,A -0.084,E1 +9.620,E3 +42.362,E4 +42.362} C_DIS
 LIN_REL {X  -9.683,Y -10.103,A +0.000,E1 +18.235,E3 +53.326,E4 +53.326} C_DIS
 LIN_REL {X  -15.230,Y -20.542,A +0.000,E1 +18.915,E3 +43.249,E4 +43.249} C_DIS
 LIN_REL {X  -10.929,Y -30.553,A +0.000,E1 +15.231,E3 +33.792,E4 +33.792} C_DIS
 LIN_REL {X  -3.920,Y -28.333,A +0.000,E1 +7.062,E3 +24.356,E4 +24.356} C_DIS
 LIN_REL {X  -0.872,Y -18.131,A +0.144,E1 +2.494,E3 +16.269,E4 +16.269} C_DIS
 LIN_REL {X  -0.134,Y -14.036,A +5.190,E1 -0.154,E3 +13.242,E4 +13.242} C_DIS
 LIN_REL {X  -0.131,Y -9.913,A +3.892,E1 -0.344,E3 +9.712,E4 +9.712} C_DIS
 LIN_REL {X  +0.026,Y -12.570,A +0.153,E1 +1.080,E3 +12.836,E4 +12.836} C_DIS
 LIN_REL {X  +0.502,Y -14.495,A +4.794,E1 -0.133,E3 +15.669,E4 +15.669} C_DIS
 LIN_REL {X  +0.735,Y -24.553,A +11.042,E1 -2.427,E3 +28.573,E4 +28.573} C_DIS
 LIN_REL {X  +0.649,Y -31.431,A +4.166,E1 -0.629,E3 +39.814,E4 +39.814} C_DIS
 LIN_REL {X  +1.404,Y -43.414,A +0.570,E1 +0.398,E3 +57.785,E4 +57.785} C_DIS
 LIN_REL {X  +1.090,Y -52.350,A +0.048,E1 +0.048,E3 +70.971,E4 +70.971} C_DIS
 LIN_REL {X  +0.308,Y -59.950,A +0.001,E1 -0.043,E3 +81.867,E4 +81.867} C_DIS
 LIN_REL {X  +0.025,Y -339.785,A +0.000,E1 -0.009,E3 +464.737,E4 +464.737} C_DIS
 LIN_REL {X  -0.018,Y -40.166,A +0.000,E1 -0.023,E3 +54.988,E4 +54.988} C_DIS
 LIN_REL {X  +0.016,Y -28.191,A +0.000,E1 -0.085,E3 +38.753,E4 +38.753} C_DIS
 LIN_REL {X  +0.081,Y -13.813,A +0.000,E1 -0.101,E3 +19.140,E4 +19.140} C_DIS
 LIN_REL {X  +0.336,Y -18.654,A +0.001,E1 -0.252,E3 +26.188,E4 +26.188} C_DIS
 LIN_REL {X  +1.707,Y -28.430,A +0.009,E1 -0.811,E3 +41.387,E4 +41.387} C_DIS
 LIN_REL {X  +5.895,Y -30.568,A +0.317,E1 -1.903,E3 +48.668,E4 +48.668} C_DIS
 LIN_REL {X  +8.493,Y -17.962,A +3.850,E1 -3.295,E3 +34.027,E4 +34.027} C_DIS
 LIN_REL {X  +6.913,Y -9.528,A +10.097,E1 -6.514,E3 +23.806,E4 +23.806} C_DIS
 LIN_REL {X  +4.348,Y -4.981,A +5.961,E1 -4.843,E3 +17.026,E4 +17.026} C_DIS
 LIN_REL {X  +5.904,Y -5.220,A +5.655,E1 -7.214,E3 +28.567,E4 +28.567} C_DIS
 LIN_REL {X  +3.104,Y -2.517,A +4.097,E1 -9.198,E3 +30.233,E4 +30.233} C_DIS
 LIN_REL {X  -1.700,Y +1.809,A +0.013,E1 -11.246,E3 +47.891,E4 +47.891} C_DIS
 LIN_REL {X  -10.267,Y +10.496,A -0.000,E1 -17.496,E3 +47.514,E4 +47.514} C_DIS
 LIN_REL {X  -12.062,Y +15.723,A -0.000,E1 -14.535,E3 +28.965,E4 +28.965} C_DIS
 LIN_REL {X  -9.261,Y +19.706,A -0.000,E1 -11.695,E3 +28.555,E4 +28.555} C_DIS
ENDFOR

HALT
LIN {X -169.488,Y 553.531,Z 0.000,A 30.000, B 0.00, C 0.00,E1 -40.759}
HALT

; PLY 19 OF 41 (Connector)

; ANGLE 51.0 (Not valid for Circ layers and non-tubes)
$APO.CDIS=85
$VEL_EXTAX[1]=100
FOR N_CYC=1 to 1
 LIN_REL {X  +0.000,Y +12.799,A +0.000,E1 -3.987,E3 +9.381,E4 +9.381} C_DIS
 LIN_REL {X  +0.000,Y +30.359,A +0.000,E1 -6.882,E3 +21.700,E4 +21.700} C_DIS
 LIN_REL {X  +0.000,Y +23.267,A -1.096,E1 -3.004,E3 +18.083,E4 +18.083} C_DIS
 LIN_REL {X  +0.000,Y +17.086,A -7.500,E1 +0.484,E3 +14.778,E4 +14.778} C_DIS
 LIN_REL {X  +0.000,Y +18.973,A -3.583,E1 -0.897,E3 +16.656,E4 +16.656} C_DIS
 LIN_REL {X  +0.000,Y +23.515,A -8.796,E1 +0.611,E3 +21.759,E4 +21.759} C_DIS
 LIN_REL {X  +0.000,Y +36.206,A -7.532,E1 +0.625,E3 +35.972,E4 +35.972} C_DIS
 LIN_REL {X  +0.000,Y +50.736,A -1.430,E1 -0.531,E3 +54.754,E4 +54.754} C_DIS
 LIN_REL {X  +0.000,Y +56.436,A -0.062,E1 -0.373,E3 +62.444,E4 +62.444} C_DIS
 LIN_REL {X  +0.000,Y +67.086,A -0.001,E1 -0.550,E3 +72.844,E4 +72.844} C_DIS
 LIN_REL {X  +0.000,Y +78.628,A +0.000,E1 -0.655,E3 +83.400,E4 +83.400} C_DIS
 LIN_REL {X  +0.000,Y +78.682,A +0.000,E1 -0.645,E3 +81.384,E4 +81.384} C_DIS
 LIN_REL {X  +0.000,Y +78.738,A -0.000,E1 -0.634,E3 +79.428,E4 +79.428} C_DIS
 LIN_REL {X  +0.000,Y +78.793,A -0.000,E1 -0.625,E3 +77.530,E4 +77.530} C_DIS
 LIN_REL {X  +0.000,Y +78.852,A -0.000,E1 -0.614,E3 +75.686,E4 +75.686} C_DIS
 LIN_REL {X  +0.000,Y +74.824,A -0.011,E1 -0.555,E3 +70.122,E4 +70.122} C_DIS
 LIN_REL {X  +0.000,Y +59.432,A -0.192,E1 -0.316,E3 +54.695,E4 +54.695} C_DIS
 LIN_REL {X  +0.000,Y +40.231,A -1.695,E1 +0.049,E3 +37.716,E4 +37.716} C_DIS
 LIN_REL {X  +0.000,Y +30.966,A -8.706,E1 +2.705,E3 +34.278,E4 +34.278} C_DIS
 LIN_REL {X  +0.000,Y +18.518,A -12.082,E1 +7.460,E3 +26.800,E4 +26.800} C_DIS
 LIN_REL {X  +0.000,Y +10.105,A -6.620,E1 +6.560,E3 +19.179,E4 +19.179} C_DIS
 LIN_REL {X  +0.000,Y +8.670,A -0.694,E1 +3.186,E3 +33.755,E4 +33.755} C_DIS
 LIN_REL {X  +0.000,Y -5.735,A +0.000,E1 +9.355,E3 +37.794,E4 +37.794} C_DIS
 LIN_REL {X  +0.000,Y -14.144,A +0.000,E1 +8.364,E3 +30.767,E4 +30.767} C_DIS
 LIN_REL {X  +0.000,Y -18.859,A +0.000,E1 +12.570,E3 +21.491,E4 +21.491} C_DIS
 LIN_REL {X  +0.000,Y -12.949,A +0.000,E1 +9.597,E3 +12.014,E4 +12.014} C_DIS
 LIN_REL {X  +0.000,Y -13.879,A +0.000,E1 +5.423,E3 +11.150,E4 +11.150} C_DIS
 LIN_REL {X  +0.000,Y -13.955,A +0.000,E1 +8.956,E3 +9.894,E4 +9.894} C_DIS
 LIN_REL {X  +0.000,Y -25.220,A +0.000,E1 +15.274,E3 +14.161,E4 +14.161} C_DIS
 LIN_REL {X  +0.000,Y -24.391,A +0.000,E1 +10.364,E3 +12.465,E4 +12.465} C_DIS
ENDFOR

HALT
LIN {X -156.443,Y 1378.736,Z 0.000,A -30.000, B 0.00, C 0.00,E1 44.416}
HALT

; PLY 20 OF 41 (Helical)

; ANGLE 51.0 (Not valid for Circ layers and non-tubes)
$APO.CDIS=85
$VEL_EXTAX[1]=100
FOR N_CYC=1 to 48
 LIN_REL {X  -9.030,Y -32.427,A +0.000,E1 +11.373,E3 +19.928,E4 +19.928} C_DIS
 LIN_REL {X  -3.428,Y -36.768,A +0.000,E1 +5.002,E3 +21.890,E4 +21.890} C_DIS
 LIN_REL {X  -0.274,Y -16.583,A +0.244,E1 +1.149,E3 +10.507,E4 +10.507} C_DIS
 LIN_REL {X  -0.016,Y -15.806,A +5.249,E1 -0.192,E3 +10.515,E4 +10.515} C_DIS
 LIN_REL {X  -0.067,Y -20.043,A +4.765,E1 +0.008,E3 +13.880,E4 +13.880} C_DIS
 LIN_REL {X  +0.458,Y -23.151,A +3.729,E1 +0.515,E3 +17.077,E4 +17.077} C_DIS
 LIN_REL {X  +0.603,Y -34.577,A +10.569,E1 -1.459,E3 +27.425,E4 +27.425} C_DIS
 LIN_REL {X  +0.027,Y -45.748,A +4.902,E1 -0.535,E3 +39.587,E4 +39.587} C_DIS
 LIN_REL {X  +0.603,Y -56.997,A +0.518,E1 +0.206,E3 +52.307,E4 +52.307} C_DIS
 LIN_REL {X  +0.425,Y -68.870,A +0.024,E1 -0.037,E3 +64.083,E4 +64.083} C_DIS
 LIN_REL {X  +0.059,Y -320.236,A +0.000,E1 -0.016,E3 +299.011,E4 +299.011} C_DIS
 LIN_REL {X  +0.069,Y -53.759,A +0.000,E1 -0.022,E3 +50.270,E4 +50.270} C_DIS
 LIN_REL {X  +0.528,Y -37.954,A +0.000,E1 -0.137,E3 +35.934,E4 +35.934} C_DIS
 LIN_REL {X  +1.417,Y -26.160,A +0.000,E1 -0.318,E3 +25.694,E4 +25.694} C_DIS
 LIN_REL {X  +1.572,Y -14.334,A +0.001,E1 -0.332,E3 +14.764,E4 +14.764} C_DIS
 LIN_REL {X  +4.266,Y -21.792,A +0.008,E1 -0.870,E3 +24.004,E4 +24.004} C_DIS
 LIN_REL {X  +11.214,Y -27.276,A +0.477,E1 -2.203,E3 +34.303,E4 +34.303} C_DIS
 LIN_REL {X  +12.317,Y -15.134,A +5.736,E1 -3.617,E3 +24.064,E4 +24.064} C_DIS
 LIN_REL {X  +11.764,Y -10.480,A +11.728,E1 -6.469,E3 +24.456,E4 +24.456} C_DIS
 LIN_REL {X  +11.997,Y -8.378,A +9.816,E1 -8.996,E3 +34.289,E4 +34.289} C_DIS
 LIN_REL {X  +5.606,Y -3.760,A +2.232,E1 -6.732,E3 +27.712,E4 +27.712} C_DIS
 LIN_REL {X  +3.237,Y -1.541,A +0.002,E1 -10.778,E3 +51.353,E4 +51.353} C_DIS
 LIN_REL {X  -6.610,Y +4.263,A -0.000,E1 -14.980,E3 +53.578,E4 +53.578} C_DIS
 LIN_REL {X  -13.406,Y +10.912,A -0.000,E1 -16.579,E3 +40.819,E4 +40.819} C_DIS
 LIN_REL {X  -17.125,Y +15.956,A -0.000,E1 -18.205,E3 +31.198,E4 +31.198} C_DIS
 LIN_REL {X  -18.335,Y +30.345,A -0.000,E1 -17.697,E3 +28.645,E4 +28.645} C_DIS
 LIN_REL {X  -8.473,Y +35.942,A -0.000,E1 -10.284,E3 +21.765,E4 +21.765} C_DIS
 LIN_REL {X  -2.079,Y +38.321,A -0.026,E1 -3.945,E3 +23.347,E4 +23.347} C_DIS
 LIN_REL {X  -0.023,Y +17.055,A -3.847,E1 -0.209,E3 +11.245,E4 +11.245} C_DIS
 LIN_REL {X  -0.076,Y +19.311,A -6.628,E1 +0.455,E3 +13.292,E4 +13.292} C_DIS
 LIN_REL {X  +0.099,Y +17.760,A -1.748,E1 -0.625,E3 +12.833,E4 +12.833} C_DIS
 LIN_REL {X  +0.575,Y +25.045,A -6.658,E1 +0.363,E3 +19.234,E4 +19.234} C_DIS
 LIN_REL {X  +0.363,Y +41.498,A -8.882,E1 +1.378,E3 +34.417,E4 +34.417} C_DIS
 LIN_REL {X  +0.365,Y +57.087,A -2.139,E1 -0.065,E3 +51.435,E4 +51.435} C_DIS
 LIN_REL {X  +0.578,Y +63.564,A -0.071,E1 -0.028,E3 +58.959,E4 +58.959} C_DIS
 LIN_REL {X  +0.161,Y +344.865,A -0.001,E1 +0.035,E3 +321.969,E4 +321.969} C_DIS
 LIN_REL {X  +0.053,Y +53.815,A -0.000,E1 +0.017,E3 +50.308,E4 +50.308} C_DIS
 LIN_REL {X  +0.420,Y +38.260,A -0.000,E1 +0.112,E3 +36.124,E4 +36.124} C_DIS
 LIN_REL {X  +1.201,Y +26.021,A -0.000,E1 +0.275,E3 +25.372,E4 +25.372} C_DIS
 LIN_REL {X  +1.408,Y +14.381,A -0.002,E1 +0.301,E3 +14.666,E4 +14.666} C_DIS
 LIN_REL {X  +3.955,Y +22.097,A -0.011,E1 +0.812,E3 +24.039,E4 +24.039} C_DIS
 LIN_REL {X  +10.721,Y +28.120,A -0.288,E1 +2.108,E3 +34.816,E4 +34.816} C_DIS
 LIN_REL {X  +10.509,Y +14.020,A -3.042,E1 +2.475,E3 +21.083,E4 +21.083} C_DIS
 LIN_REL {X  +10.897,Y +10.324,A -11.202,E1 +5.715,E3 +21.337,E4 +21.337} C_DIS
 LIN_REL {X  +8.885,Y +7.105,A -7.308,E1 +5.085,E3 +21.171,E4 +21.171} C_DIS
 LIN_REL {X  +9.335,Y +6.223,A -7.404,E1 +8.560,E3 +31.328,E4 +31.328} C_DIS
 LIN_REL {X  +5.127,Y +3.378,A -0.743,E1 +6.995,E3 +33.252,E4 +33.252} C_DIS
 LIN_REL {X  +0.448,Y -0.281,A -0.000,E1 +13.217,E3 +54.715,E4 +54.715} C_DIS
 LIN_REL {X  -9.943,Y -6.919,A -0.000,E1 +14.958,E3 +52.086,E4 +52.086} C_DIS
 LIN_REL {X  -14.285,Y -11.577,A -0.000,E1 +17.691,E3 +34.806,E4 +34.806} C_DIS
 LIN_REL {X  -28.092,Y -35.117,A -0.000,E1 +26.525,E3 +44.941,E4 +44.941} C_DIS
ENDFOR

HALT
LIN {X -169.926,Y 1383.166,Z 0.000,A -30.000, B 0.00, C 0.00,E1 46.229}
HALT

; PLY 21 OF 41 (Connector)

; ANGLE 51.0 (Not valid for Circ layers and non-tubes)
$APO.CDIS=85
$VEL_EXTAX[1]=100
FOR N_CYC=1 to 1
 LIN_REL {X  +0.000,Y -12.602,A +0.000,E1 +3.784,E3 +6.932,E4 +6.932} C_DIS
 LIN_REL {X  +0.000,Y -27.216,A +0.000,E1 +6.525,E3 +14.401,E4 +14.401} C_DIS
 LIN_REL {X  +0.000,Y -38.785,A +0.000,E1 +4.264,E3 +23.371,E4 +23.371} C_DIS
 LIN_REL {X  +0.000,Y -24.065,A +1.457,E1 +0.871,E3 +16.025,E4 +16.025} C_DIS
 LIN_REL {X  +0.000,Y -19.790,A +7.637,E1 -0.455,E3 +14.007,E4 +14.007} C_DIS
 LIN_REL {X  +0.000,Y -24.148,A +4.306,E1 +0.403,E3 +18.029,E4 +18.029} C_DIS
 LIN_REL {X  +0.000,Y -38.172,A +10.312,E1 -1.377,E3 +31.128,E4 +31.128} C_DIS
 LIN_REL {X  +0.000,Y -38.550,A +5.420,E1 -0.767,E3 +35.071,E4 +35.071} C_DIS
 LIN_REL {X  +0.000,Y -47.507,A +0.787,E1 -0.162,E3 +45.102,E4 +45.102} C_DIS
 LIN_REL {X  +0.000,Y -538.009,A +0.082,E1 -0.089,E3 +513.437,E4 +513.437} C_DIS
 LIN_REL {X  +0.000,Y -35.041,A +0.012,E1 -0.036,E3 +33.460,E4 +33.460} C_DIS
 LIN_REL {X  +0.000,Y -20.023,A +0.033,E1 -0.041,E3 +19.146,E4 +19.146} C_DIS
 LIN_REL {X  +0.000,Y -18.719,A +0.101,E1 -0.050,E3 +17.960,E4 +17.960} C_DIS
 LIN_REL {X  +0.000,Y -30.540,A +0.798,E1 -0.137,E3 +29.833,E4 +29.833} C_DIS
 LIN_REL {X  +0.000,Y -33.173,A +5.212,E1 -1.496,E3 +36.376,E4 +36.376} C_DIS
 LIN_REL {X  +0.000,Y -23.920,A +13.673,E1 -7.747,E3 +34.806,E4 +34.806} C_DIS
 LIN_REL {X  +0.000,Y -10.569,A +9.309,E1 -8.244,E3 +22.389,E4 +22.389} C_DIS
 LIN_REL {X  +0.000,Y -5.110,A +0.861,E1 -4.351,E3 +32.624,E4 +32.624} C_DIS
 LIN_REL {X  +0.000,Y +10.810,A -0.000,E1 -12.601,E3 +46.456,E4 +46.456} C_DIS
 LIN_REL {X  +0.000,Y +18.529,A -0.000,E1 -10.649,E3 +27.770,E4 +27.770} C_DIS
 LIN_REL {X  +0.000,Y +24.692,A -0.000,E1 -16.991,E3 +24.277,E4 +24.277} C_DIS
 LIN_REL {X  +0.000,Y +25.767,A -0.000,E1 -14.337,E3 +19.576,E4 +19.576} C_DIS
 LIN_REL {X  +0.000,Y +20.656,A -0.000,E1 -12.326,E3 +12.615,E4 +12.615} C_DIS
 LIN_REL {X  +0.000,Y +19.416,A -0.000,E1 -8.493,E3 +10.792,E4 +10.792} C_DIS
ENDFOR

HALT
LIN {X -154.967,Y 537.023,Z 0.000,A 30.000, B 0.00, C 0.00,E1 -42.595}
HALT

; PLY 22 OF 41 (Helical)

; ANGLE 51.0 (Not valid for Circ layers and non-tubes)
$APO.CDIS=85
$VEL_EXTAX[1]=100
FOR N_CYC=1 to 48
 LIN_REL {X  -10.811,Y +36.260,A +0.000,E1 -12.416,E3 +27.947,E4 +27.947} C_DIS
 LIN_REL {X  -3.577,Y +40.091,A +0.000,E1 -5.224,E3 +25.966,E4 +25.966} C_DIS
 LIN_REL {X  -0.219,Y +18.824,A -1.163,E1 -0.968,E3 +12.722,E4 +12.722} C_DIS
 LIN_REL {X  -0.050,Y +21.563,A -7.599,E1 +0.467,E3 +15.352,E4 +15.352} C_DIS
 LIN_REL {X  +0.171,Y +24.743,A -4.681,E1 -0.410,E3 +18.733,E4 +18.733} C_DIS
 LIN_REL {X  +0.616,Y +31.428,A -8.957,E1 +0.950,E3 +25.710,E4 +25.710} C_DIS
 LIN_REL {X  +0.290,Y +46.981,A -6.719,E1 +0.946,E3 +41.995,E4 +41.995} C_DIS
 LIN_REL {X  +0.659,Y +57.229,A -0.855,E1 -0.137,E3 +54.563,E4 +54.563} C_DIS
 LIN_REL {X  +0.490,Y +68.534,A -0.026,E1 +0.020,E3 +66.375,E4 +66.375} C_DIS
 LIN_REL {X  +0.084,Y +327.243,A -0.000,E1 +0.020,E3 +318.155,E4 +318.155} C_DIS
 LIN_REL {X  +0.058,Y +53.764,A -0.000,E1 +0.022,E3 +52.341,E4 +52.341} C_DIS
 LIN_REL {X  +0.446,Y +38.100,A -0.000,E1 +0.131,E3 +37.488,E4 +37.488} C_DIS
 LIN_REL {X  +1.180,Y +25.289,A -0.001,E1 +0.292,E3 +25.683,E4 +25.683} C_DIS
 LIN_REL {X  +1.254,Y +13.058,A -0.002,E1 +0.286,E3 +13.825,E4 +13.825} C_DIS
 LIN_REL {X  +3.107,Y +19.116,A -0.013,E1 +0.673,E3 +21.324,E4 +21.324} C_DIS
 LIN_REL {X  +9.300,Y +27.905,A -0.238,E1 +1.897,E3 +34.779,E4 +34.779} C_DIS
 LIN_REL {X  +11.420,Y +17.057,A -3.115,E1 +2.743,E3 +25.538,E4 +25.538} C_DIS
 LIN_REL {X  +11.028,Y +10.972,A -11.189,E1 +5.880,E3 +22.820,E4 +22.820} C_DIS
 LIN_REL {X  +12.521,Y +9.722,A -10.950,E1 +8.685,E3 +33.772,E4 +33.772} C_DIS
 LIN_REL {X  +7.374,Y +4.849,A -4.342,E1 +8.310,E3 +32.797,E4 +32.797} C_DIS
 LIN_REL {X  +3.832,Y +2.241,A -0.150,E1 +11.634,E3 +53.883,E4 +53.883} C_DIS
 LIN_REL {X  -7.399,Y -4.859,A +0.000,E1 +16.271,E3 +58.373,E4 +58.373} C_DIS
 LIN_REL {X  -14.203,Y -11.097,A +0.000,E1 +18.114,E3 +42.644,E4 +42.644} C_DIS
 LIN_REL {X  -18.689,Y -19.556,A +0.000,E1 +18.681,E3 +36.627,E4 +36.627} C_DIS
 LIN_REL {X  -15.212,Y -31.042,A +0.000,E1 +15.502,E3 +30.141,E4 +30.141} C_DIS
 LIN_REL {X  -7.287,Y -41.504,A +0.000,E1 +8.924,E3 +27.729,E4 +27.729} C_DIS
 LIN_REL {X  -0.961,Y -26.173,A +0.078,E1 +2.132,E3 +17.117,E4 +17.117} C_DIS
 LIN_REL {X  -0.064,Y -13.198,A +2.454,E1 +0.261,E3 +9.061,E4 +9.061} C_DIS
 LIN_REL {X  -0.057,Y -22.797,A +7.104,E1 -0.275,E3 +16.348,E4 +16.348} C_DIS
 LIN_REL {X  +0.442,Y -26.354,A +5.138,E1 +0.368,E3 +20.249,E4 +20.249} C_DIS
 LIN_REL {X  +0.562,Y -36.469,A +10.649,E1 -1.545,E3 +30.410,E4 +30.410} C_DIS
 LIN_REL {X  +0.175,Y -47.247,A +4.171,E1 -0.381,E3 +43.126,E4 +43.126} C_DIS
 LIN_REL {X  +0.741,Y -59.210,A +0.388,E1 +0.140,E3 +56.779,E4 +56.779} C_DIS
 LIN_REL {X  +0.381,Y -69.504,A +0.018,E1 -0.039,E3 +67.374,E4 +67.374} C_DIS
 LIN_REL {X  +0.050,Y -316.689,A +0.000,E1 -0.013,E3 +307.825,E4 +307.825} C_DIS
 LIN_REL {X  +0.074,Y -53.717,A +0.000,E1 -0.028,E3 +52.299,E4 +52.299} C_DIS
 LIN_REL {X  +0.544,Y -37.828,A +0.000,E1 -0.154,E3 +37.302,E4 +37.302} C_DIS
 LIN_REL {X  +1.344,Y -25.044,A +0.001,E1 -0.325,E3 +25.580,E4 +25.580} C_DIS
 LIN_REL {X  +1.437,Y -13.433,A +0.001,E1 -0.322,E3 +14.344,E4 +14.344} C_DIS
 LIN_REL {X  +2.665,Y -15.721,A +0.007,E1 -0.573,E3 +17.621,E4 +17.621} C_DIS
 LIN_REL {X  +8.198,Y -25.603,A +0.196,E1 -1.674,E3 +31.655,E4 +31.655} C_DIS
 LIN_REL {X  +11.248,Y -17.972,A +2.757,E1 -2.657,E3 +26.284,E4 +26.284} C_DIS
 LIN_REL {X  +11.364,Y -11.650,A +10.503,E1 -5.617,E3 +23.425,E4 +23.425} C_DIS
 LIN_REL {X  +12.920,Y -10.078,A +11.389,E1 -8.617,E3 +33.602,E4 +33.602} C_DIS
 LIN_REL {X  +6.700,Y -4.434,A +5.070,E1 -7.345,E3 +26.447,E4 +26.447} C_DIS
 LIN_REL {X  +4.769,Y -2.981,A +0.076,E1 -8.796,E3 +43.543,E4 +43.543} C_DIS
 LIN_REL {X  -3.270,Y +2.369,A -0.000,E1 -15.141,E3 +57.165,E4 +57.165} C_DIS
 LIN_REL {X  -13.746,Y +10.257,A -0.000,E1 -18.528,E3 +52.019,E4 +52.019} C_DIS
 LIN_REL {X  -31.899,Y +36.565,A -0.000,E1 -32.164,E3 +62.310,E4 +62.310} C_DIS
ENDFOR

HALT
LIN {X -170.370,Y 532.350,Z 0.000,A 30.000, B 0.00, C 0.00,E1 -44.710}
HALT

; PLY 23 OF 41 (Connector)

; ANGLE 51.0 (Not valid for Circ layers and non-tubes)
$APO.CDIS=85
$VEL_EXTAX[1]=100
FOR N_CYC=1 to 1
 LIN_REL {X  +0.000,Y +15.029,A +0.000,E1 -4.321,E3 +12.189,E4 +12.189} C_DIS
 LIN_REL {X  +0.000,Y +6.220,A +0.000,E1 -1.601,E3 +4.697,E4 +4.697} C_DIS
 LIN_REL {X  +0.000,Y +24.653,A +0.000,E1 -5.126,E3 +17.489,E4 +17.489} C_DIS
 LIN_REL {X  +0.000,Y +37.708,A -0.009,E1 -3.415,E3 +27.700,E4 +27.700} C_DIS
 LIN_REL {X  +0.000,Y +19.328,A -3.663,E1 -0.152,E3 +15.211,E4 +15.211} C_DIS
 LIN_REL {X  +0.000,Y +23.916,A -8.075,E1 +0.838,E3 +20.332,E4 +20.332} C_DIS
 LIN_REL {X  +0.000,Y +31.626,A -10.115,E1 +1.424,E3 +30.452,E4 +30.452} C_DIS
 LIN_REL {X  +0.000,Y +39.224,A -7.179,E1 +2.544,E3 +45.867,E4 +45.867} C_DIS
 LIN_REL {X  +0.000,Y +46.975,A -0.908,E1 +1.007,E3 +58.860,E4 +58.860} C_DIS
 LIN_REL {X  +0.000,Y +55.211,A -0.050,E1 +0.944,E3 +70.734,E4 +70.734} C_DIS
 LIN_REL {X  +0.000,Y +64.963,A -0.001,E1 +1.042,E3 +86.064,E4 +86.064} C_DIS
 LIN_REL {X  +0.000,Y +67.929,A +0.000,E1 +1.107,E3 +93.423,E4 +93.423} C_DIS
 LIN_REL {X  +0.000,Y +67.993,A +0.000,E1 +1.142,E3 +97.259,E4 +97.259} C_DIS
 LIN_REL {X  +0.000,Y +65.324,A -0.000,E1 +1.133,E3 +97.225,E4 +97.225} C_DIS
 LIN_REL {X  +0.000,Y +62.642,A -0.000,E1 +1.122,E3 +96.966,E4 +96.966} C_DIS
 LIN_REL {X  +0.000,Y +62.666,A -0.000,E1 +1.163,E3 +100.948,E4 +100.948} C_DIS
 LIN_REL {X  +0.000,Y +59.744,A -0.007,E1 +1.177,E3 +100.215,E4 +100.215} C_DIS
 LIN_REL {X  +0.000,Y +49.505,A -0.086,E1 +1.180,E3 +86.291,E4 +86.291} C_DIS
 LIN_REL {X  +0.000,Y +36.035,A -0.515,E1 +1.199,E3 +64.973,E4 +64.973} C_DIS
 LIN_REL {X  +0.000,Y +25.348,A -2.937,E1 +1.794,E3 +47.058,E4 +47.058} C_DIS
 LIN_REL {X  +0.000,Y +17.431,A -10.020,E1 +7.261,E3 +37.409,E4 +37.409} C_DIS
 LIN_REL {X  +0.000,Y +10.135,A -11.903,E1 +13.527,E3 +32.265,E4 +32.265} C_DIS
 LIN_REL {X  +0.000,Y +4.120,A -4.488,E1 +10.183,E3 +33.393,E4 +33.393} C_DIS
 LIN_REL {X  +0.000,Y -6.819,A -0.044,E1 +12.263,E3 +46.162,E4 +46.162} C_DIS
 LIN_REL {X  +0.000,Y -19.596,A +0.000,E1 +14.850,E3 +42.275,E4 +42.275} C_DIS
 LIN_REL {X  +0.000,Y -15.074,A +0.000,E1 +9.183,E3 +22.183,E4 +22.183} C_DIS
ENDFOR

HALT
LIN {X -162.795,Y 1362.741,Z 0.000,A -30.000, B 0.00, C 0.00,E1 34.081}
HALT

; PLY 24 OF 41 (Helical)

; ANGLE 51.0 (Not valid for Circ layers and non-tubes)
$APO.CDIS=85
$VEL_EXTAX[1]=100
FOR N_CYC=1 to 35
 LIN_REL {X  -4.501,Y -25.542,A +0.000,E1 +9.037,E3 +34.380,E4 +34.380} C_DIS
 LIN_REL {X  -1.914,Y -22.618,A +0.265,E1 +4.169,E3 +26.307,E4 +26.307} C_DIS
 LIN_REL {X  -0.511,Y -18.809,A +6.136,E1 +0.292,E3 +22.787,E4 +22.787} C_DIS
 LIN_REL {X  +0.370,Y -24.467,A +8.422,E1 -0.171,E3 +32.330,E4 +32.330} C_DIS
 LIN_REL {X  +1.096,Y -26.677,A +11.106,E1 -2.737,E3 +39.552,E4 +39.552} C_DIS
 LIN_REL {X  +1.778,Y -35.064,A +3.580,E1 -0.390,E3 +56.808,E4 +56.808} C_DIS
 LIN_REL {X  +2.268,Y -42.918,A +0.436,E1 +0.469,E3 +72.386,E4 +72.386} C_DIS
 LIN_REL {X  +1.487,Y -51.473,A +0.052,E1 +0.149,E3 +88.344,E4 +88.344} C_DIS
 LIN_REL {X  +0.468,Y -59.770,A +0.003,E1 -0.016,E3 +103.397,E4 +103.397} C_DIS
 LIN_REL {X  +0.053,Y -302.335,A +0.000,E1 -0.009,E3 +524.096,E4 +524.096} C_DIS
 LIN_REL {X  -0.084,Y -60.320,A +0.000,E1 -0.028,E3 +104.637,E4 +104.637} C_DIS
 LIN_REL {X  -0.481,Y -55.891,A +0.002,E1 -0.258,E3 +97.456,E4 +97.456} C_DIS
 LIN_REL {X  -0.190,Y -44.219,A +0.033,E1 -0.950,E3 +78.992,E4 +78.992} C_DIS
 LIN_REL {X  +2.396,Y -31.599,A +0.368,E1 -1.747,E3 +60.215,E4 +60.215} C_DIS
 LIN_REL {X  +5.252,Y -20.789,A +2.646,E1 -2.990,E3 +44.719,E4 +44.719} C_DIS
 LIN_REL {X  +5.658,Y -12.412,A +9.194,E1 -7.032,E3 +34.006,E4 +34.006} C_DIS
 LIN_REL {X  +5.280,Y -8.436,A +10.499,E1 -10.641,E3 +36.620,E4 +36.620} C_DIS
 LIN_REL {X  +2.282,Y -2.574,A +6.733,E1 -9.487,E3 +25.893,E4 +25.893} C_DIS
 LIN_REL {X  -0.258,Y +0.586,A +0.525,E1 -9.592,E3 +40.594,E4 +40.594} C_DIS
 LIN_REL {X  -7.391,Y +11.165,A -0.000,E1 -16.300,E3 +53.039,E4 +53.039} C_DIS
 LIN_REL {X  -10.753,Y +24.532,A -0.000,E1 -17.528,E3 +48.774,E4 +48.774} C_DIS
 LIN_REL {X  -6.627,Y +29.273,A -0.000,E1 -11.351,E3 +37.267,E4 +37.267} C_DIS
 LIN_REL {X  -2.001,Y +22.736,A -0.248,E1 -4.264,E3 +26.307,E4 +26.307} C_DIS
 LIN_REL {X  -0.509,Y +17.062,A -5.553,E1 -0.282,E3 +20.616,E4 +20.616} C_DIS
 LIN_REL {X  +0.053,Y +21.360,A -7.381,E1 +0.095,E3 +27.929,E4 +27.929} C_DIS
 LIN_REL {X  +0.927,Y +23.668,A -9.901,E1 +2.004,E3 +34.269,E4 +34.269} C_DIS
 LIN_REL {X  +1.023,Y +21.795,A -4.895,E1 +1.160,E3 +34.177,E4 +34.177} C_DIS
 LIN_REL {X  +1.632,Y +29.275,A -1.661,E1 -0.088,E3 +48.162,E4 +48.162} C_DIS
 LIN_REL {X  +1.911,Y +37.733,A -0.323,E1 -0.355,E3 +63.808,E4 +63.808} C_DIS
 LIN_REL {X  +1.313,Y +45.921,A -0.036,E1 -0.136,E3 +78.811,E4 +78.811} C_DIS
 LIN_REL {X  +0.497,Y +56.831,A -0.002,E1 +0.012,E3 +98.268,E4 +98.268} C_DIS
 LIN_REL {X  +0.070,Y +308.121,A -0.000,E1 +0.011,E3 +534.042,E4 +534.042} C_DIS
 LIN_REL {X  -0.082,Y +60.329,A -0.000,E1 +0.027,E3 +104.637,E4 +104.637} C_DIS
 LIN_REL {X  -0.491,Y +55.923,A -0.003,E1 +0.255,E3 +97.487,E4 +97.487} C_DIS
 LIN_REL {X  -0.264,Y +44.278,A -0.042,E1 +0.946,E3 +79.036,E4 +79.036} C_DIS
 LIN_REL {X  +2.366,Y +31.519,A -0.302,E1 +1.724,E3 +60.017,E4 +60.017} C_DIS
 LIN_REL {X  +5.330,Y +20.740,A -2.329,E1 +2.792,E3 +44.464,E4 +44.464} C_DIS
 LIN_REL {X  +5.850,Y +12.616,A -9.701,E1 +7.315,E3 +34.567,E4 +34.567} C_DIS
 LIN_REL {X  +4.787,Y +7.877,A -10.732,E1 +10.514,E3 +33.500,E4 +33.500} C_DIS
 LIN_REL {X  +2.568,Y +3.023,A -6.482,E1 +9.771,E3 +29.132,E4 +29.132} C_DIS
 LIN_REL {X  -0.251,Y -0.622,A -0.409,E1 +9.299,E3 +39.844,E4 +39.844} C_DIS
 LIN_REL {X  -7.167,Y -10.489,A +0.000,E1 +16.099,E3 +52.628,E4 +52.628} C_DIS
 LIN_REL {X  -8.237,Y -16.267,A +0.000,E1 +12.726,E3 +28.365,E4 +28.365} C_DIS
 LIN_REL {X  -5.003,Y -13.072,A +0.000,E1 +7.486,E3 +24.478,E4 +24.478} C_DIS
ENDFOR

HALT
LIN {X -170.809,Y 1361.495,Z 0.000,A -30.000, B 0.00, C 0.00,E1 36.738}
HALT

; PLY 25 OF 41 (Connector)

; ANGLE 51.0 (Not valid for Circ layers and non-tubes)
$APO.CDIS=85
$VEL_EXTAX[1]=100
FOR N_CYC=1 to 1
 LIN_REL {X  +0.000,Y -16.436,A +0.000,E1 +4.766,E3 +18.189,E4 +18.189} C_DIS
 LIN_REL {X  +0.000,Y -27.982,A +0.000,E1 +6.082,E3 +28.578,E4 +28.578} C_DIS
 LIN_REL {X  +0.000,Y -17.864,A +2.599,E1 +1.517,E3 +18.513,E4 +18.513} C_DIS
 LIN_REL {X  +0.000,Y -20.115,A +7.696,E1 +0.209,E3 +21.787,E4 +21.787} C_DIS
 LIN_REL {X  +0.000,Y -29.842,A +10.763,E1 -0.903,E3 +34.869,E4 +34.869} C_DIS
 LIN_REL {X  +0.000,Y -29.870,A +6.910,E1 -0.661,E3 +36.705,E4 +36.705} C_DIS
 LIN_REL {X  +0.000,Y -42.152,A +1.743,E1 +1.273,E3 +50.979,E4 +50.979} C_DIS
 LIN_REL {X  +0.000,Y -53.535,A +0.252,E1 +1.989,E3 +61.077,E4 +61.077} C_DIS
 LIN_REL {X  +0.000,Y -63.220,A +0.035,E1 +2.348,E3 +66.289,E4 +66.289} C_DIS
 LIN_REL {X  +0.000,Y -78.452,A +0.002,E1 +2.750,E3 +74.316,E4 +74.316} C_DIS
 LIN_REL {X  +0.000,Y -82.906,A -0.000,E1 +2.685,E3 +70.060,E4 +70.060} C_DIS
 LIN_REL {X  +0.000,Y -87.685,A -0.000,E1 +2.622,E3 +65.727,E4 +65.727} C_DIS
 LIN_REL {X  +0.000,Y -89.414,A +0.000,E1 +2.474,E3 +59.125,E4 +59.125} C_DIS
 LIN_REL {X  +0.000,Y -91.630,A +0.000,E1 +2.349,E3 +53.149,E4 +53.149} C_DIS
 LIN_REL {X  +0.000,Y -94.419,A +0.000,E1 +2.243,E3 +47.640,E4 +47.640} C_DIS
 LIN_REL {X  +0.000,Y -92.480,A +0.022,E1 +2.026,E3 +40.394,E4 +40.394} C_DIS
 LIN_REL {X  +0.000,Y -77.505,A +0.361,E1 +1.515,E3 +30.832,E4 +30.832} C_DIS
 LIN_REL {X  +0.000,Y -62.833,A +2.339,E1 +0.404,E3 +31.130,E4 +31.130} C_DIS
 LIN_REL {X  +0.000,Y -46.115,A +6.054,E1 -0.904,E3 +31.809,E4 +31.809} C_DIS
 LIN_REL {X  +0.000,Y -30.365,A +10.891,E1 -3.009,E3 +28.206,E4 +28.206} C_DIS
 LIN_REL {X  +0.000,Y -14.037,A +8.631,E1 -3.537,E3 +17.834,E4 +17.834} C_DIS
 LIN_REL {X  +0.000,Y -12.075,A +1.702,E1 -1.597,E3 +28.985,E4 +28.985} C_DIS
 LIN_REL {X  +0.000,Y +2.397,A -0.000,E1 -0.722,E3 +24.325,E4 +24.325} C_DIS
 LIN_REL {X  +0.000,Y +23.417,A -0.000,E1 -4.058,E3 +36.450,E4 +36.450} C_DIS
 LIN_REL {X  +0.000,Y +41.228,A -0.000,E1 -6.736,E3 +34.008,E4 +34.008} C_DIS
 LIN_REL {X  +0.000,Y +26.775,A -0.000,E1 -4.301,E3 +15.752,E4 +15.752} C_DIS
 LIN_REL {X  +0.000,Y +17.676,A -0.000,E1 -0.018,E3 +8.815,E4 +8.815} C_DIS
 LIN_REL {X  +0.000,Y +17.690,A -0.000,E1 -4.806,E3 +8.011,E4 +8.011} C_DIS
 LIN_REL {X  +0.000,Y +27.071,A -0.000,E1 -14.519,E3 +11.254,E4 +11.254} C_DIS
 LIN_REL {X  +0.000,Y +32.178,A -0.000,E1 -18.181,E3 +11.845,E4 +11.845} C_DIS
 LIN_REL {X  +0.000,Y +25.924,A -0.000,E1 -21.603,E3 +8.333,E4 +8.333} C_DIS
 LIN_REL {X  +0.000,Y +11.068,A -0.000,E1 -11.450,E3 +3.262,E4 +3.262} C_DIS
 LIN_REL {X  +0.000,Y +0.739,A -0.000,E1 +1.238,E3 +0.253,E4 +0.253} C_DIS
 LIN_REL {X  +0.000,Y -2.102,A -0.000,E1 +15.704,E3 +0.118,E4 +0.118} C_DIS
 LIN_REL {X  +0.000,Y -2.659,A -0.000,E1 +3.851,E3 +0.050,E4 +0.050} C_DIS
 LIN_REL {X  +0.000,Y +0.385,A -0.000,E1 -6.623,E3 +0.050,E4 +0.050} C_DIS
 LIN_REL {X  +0.000,Y +13.743,A -0.000,E1 -4.018,E3 +3.714,E4 +3.714} C_DIS
 LIN_REL {X  +0.000,Y +17.738,A -0.000,E1 -13.587,E3 +4.217,E4 +4.217} C_DIS
 LIN_REL {X  +0.000,Y +23.461,A -0.000,E1 -16.495,E3 +4.847,E4 +4.847} C_DIS
 LIN_REL {X  +0.000,Y +12.900,A -0.000,E1 -8.145,E3 +2.201,E4 +2.201} C_DIS
 LIN_REL {X  +0.000,Y +2.960,A -0.000,E1 -0.283,E3 +0.607,E4 +0.607} C_DIS
 LIN_REL {X  +0.000,Y -8.613,A -0.000,E1 +8.261,E3 +0.174,E4 +0.174} C_DIS
 LIN_REL {X  +0.000,Y -6.051,A -0.000,E1 +1.135,E3 +0.117,E4 +0.117} C_DIS
 LIN_REL {X  +0.000,Y +13.428,A -0.000,E1 -8.408,E3 +7.151,E4 +7.151} C_DIS
 LIN_REL {X  +0.000,Y +18.093,A -0.000,E1 -6.272,E3 +7.091,E4 +7.091} C_DIS
ENDFOR

HALT
LIN {X -151.416,Y 528.607,Z 0.000,A 30.000, B 0.00, C 0.00,E1 -58.466}
HALT

; PLY 26 OF 41 (Helical)

; ANGLE 51.0 (Not valid for Circ layers and non-tubes)
$APO.CDIS=85
$VEL_EXTAX[1]=100
FOR N_CYC=1 to 57
 LIN_REL {X  -7.683,Y +15.619,A +0.000,E1 -4.333,E3 +12.343,E4 +12.343} C_DIS
 LIN_REL {X  -6.216,Y +22.423,A +0.000,E1 -5.411,E3 +8.124,E4 +8.124} C_DIS
 LIN_REL {X  -4.547,Y +41.423,A +0.000,E1 -3.687,E3 +13.503,E4 +13.503} C_DIS
 LIN_REL {X  -0.790,Y +34.064,A -0.281,E1 -1.031,E3 +11.991,E4 +11.991} C_DIS
 LIN_REL {X  +0.013,Y +21.319,A -5.522,E1 +0.050,E3 +7.960,E4 +7.960} C_DIS
 LIN_REL {X  +0.079,Y +35.049,A -6.770,E1 +0.017,E3 +13.532,E4 +13.532} C_DIS
 LIN_REL {X  +0.532,Y +50.371,A -6.060,E1 -0.171,E3 +20.516,E4 +20.516} C_DIS
 LIN_REL {X  +0.342,Y +67.828,A -7.560,E1 +0.578,E3 +29.488,E4 +29.488} C_DIS
 LIN_REL {X  -0.487,Y +82.582,A -3.492,E1 +0.108,E3 +39.130,E4 +39.130} C_DIS
 LIN_REL {X  +0.048,Y +97.020,A -0.314,E1 -0.046,E3 +48.916,E4 +48.916} C_DIS
 LIN_REL {X  +0.037,Y +176.085,A -0.001,E1 +0.010,E3 +89.242,E4 +89.242} C_DIS
 LIN_REL {X  +0.051,Y +79.115,A -0.000,E1 +0.007,E3 +40.146,E4 +40.146} C_DIS
 LIN_REL {X  +1.122,Y +63.804,A -0.000,E1 +0.131,E3 +33.231,E4 +33.231} C_DIS
 LIN_REL {X  +6.093,Y +47.227,A -0.000,E1 +0.668,E3 +28.561,E4 +28.561} C_DIS
 LIN_REL {X  +13.995,Y +34.566,A -0.022,E1 +1.662,E3 +26.969,E4 +26.969} C_DIS
 LIN_REL {X  +11.280,Y +14.444,A -0.612,E1 +1.470,E3 +13.301,E4 +13.301} C_DIS
 LIN_REL {X  +16.166,Y +13.163,A -8.011,E1 +3.173,E3 +15.145,E4 +15.145} C_DIS
 LIN_REL {X  +21.542,Y +14.922,A -13.356,E1 +6.204,E3 +27.096,E4 +27.096} C_DIS
 LIN_REL {X  +13.285,Y +20.568,A -7.085,E1 +6.936,E3 +39.984,E4 +39.984} C_DIS
 LIN_REL {X  +5.030,Y +26.809,A -0.914,E1 +7.056,E3 +57.725,E4 +57.725} C_DIS
 LIN_REL {X  -1.660,Y +14.124,A +0.000,E1 +4.866,E3 +45.473,E4 +45.473} C_DIS
 LIN_REL {X  -0.559,Y -3.695,A +0.000,E1 +5.771,E3 +37.672,E4 +37.672} C_DIS
 LIN_REL {X  +0.122,Y -20.795,A +0.000,E1 +15.516,E3 +38.747,E4 +38.747} C_DIS
 LIN_REL {X  -0.972,Y -18.987,A +0.000,E1 +14.059,E3 +24.260,E4 +24.260} C_DIS
 LIN_REL {X  -7.519,Y -13.404,A +0.000,E1 +9.775,E3 +24.095,E4 +24.095} C_DIS
 LIN_REL {X  -15.218,Y -10.688,A +0.000,E1 +19.831,E3 +23.681,E4 +23.681} C_DIS
 LIN_REL {X  -9.136,Y -5.630,A +0.000,E1 +8.459,E3 +11.070,E4 +11.070} C_DIS
 LIN_REL {X  -13.057,Y -10.496,A +0.000,E1 +9.302,E3 +19.019,E4 +19.019} C_DIS
 LIN_REL {X  -17.624,Y -20.051,A +0.000,E1 +14.042,E3 +20.394,E4 +20.394} C_DIS
 LIN_REL {X  -9.962,Y -16.006,A +0.000,E1 +5.647,E3 +12.442,E4 +12.442} C_DIS
 LIN_REL {X  -6.685,Y -20.348,A +0.000,E1 +4.812,E3 +9.318,E4 +9.318} C_DIS
 LIN_REL {X  -5.736,Y -41.006,A +0.000,E1 +4.607,E3 +13.196,E4 +13.196} C_DIS
 LIN_REL {X  -1.108,Y -34.565,A +0.028,E1 +1.193,E3 +11.922,E4 +11.922} C_DIS
 LIN_REL {X  -0.024,Y -19.959,A +3.838,E1 +0.090,E3 +7.362,E4 +7.362} C_DIS
 LIN_REL {X  +0.048,Y -31.874,A +6.931,E1 -0.053,E3 +12.145,E4 +12.145} C_DIS
 LIN_REL {X  +0.368,Y -36.657,A +4.418,E1 +0.284,E3 +14.593,E4 +14.593} C_DIS
 LIN_REL {X  +0.577,Y -50.902,A +6.996,E1 -0.315,E3 +21.321,E4 +21.321} C_DIS
 LIN_REL {X  -0.124,Y -69.571,A +5.974,E1 -0.533,E3 +31.093,E4 +31.093} C_DIS
 LIN_REL {X  -0.430,Y -86.405,A +1.739,E1 +0.115,E3 +42.194,E4 +42.194} C_DIS
 LIN_REL {X  +0.121,Y -97.701,A +0.076,E1 -0.006,E3 +49.382,E4 +49.382} C_DIS
 LIN_REL {X  +0.013,Y -151.477,A -0.000,E1 -0.004,E3 +76.676,E4 +76.676} C_DIS
 LIN_REL {X  +0.077,Y -79.107,A +0.000,E1 -0.010,E3 +40.108,E4 +40.108} C_DIS
 LIN_REL {X  +1.594,Y -64.321,A +0.000,E1 -0.185,E3 +33.831,E4 +33.831} C_DIS
 LIN_REL {X  +7.395,Y -46.433,A +0.000,E1 -0.816,E3 +29.076,E4 +29.076} C_DIS
 LIN_REL {X  +14.108,Y -31.004,A +0.037,E1 -1.707,E3 +24.960,E4 +24.960} C_DIS
 LIN_REL {X  +13.809,Y -15.583,A +1.938,E1 -1.920,E3 +14.819,E4 +14.819} C_DIS
 LIN_REL {X  +17.872,Y -13.335,A +10.995,E1 -4.101,E3 +17.426,E4 +17.426} C_DIS
 LIN_REL {X  +19.115,Y -14.796,A +11.317,E1 -6.107,E3 +28.649,E4 +28.649} C_DIS
 LIN_REL {X  +11.626,Y -22.627,A +5.471,E1 -7.271,E3 +44.756,E4 +44.756} C_DIS
 LIN_REL {X  +3.173,Y -23.870,A +0.242,E1 -6.236,E3 +53.703,E4 +53.703} C_DIS
 LIN_REL {X  -1.814,Y -11.128,A -0.000,E1 -4.041,E3 +38.125,E4 +38.125} C_DIS
 LIN_REL {X  -0.708,Y +1.526,A -0.000,E1 -3.919,E3 +28.029,E4 +28.029} C_DIS
 LIN_REL {X  +0.328,Y +15.564,A -0.000,E1 -10.727,E3 +35.129,E4 +35.129} C_DIS
 LIN_REL {X  -0.462,Y +19.075,A -0.000,E1 -15.669,E3 +26.400,E4 +26.400} C_DIS
 LIN_REL {X  -3.761,Y +16.992,A -0.000,E1 -9.585,E3 +23.615,E4 +23.615} C_DIS
 LIN_REL {X  -13.018,Y +11.098,A -0.000,E1 -16.467,E3 +24.914,E4 +24.914} C_DIS
 LIN_REL {X  -12.771,Y +8.176,A -0.000,E1 -14.705,E3 +16.405,E4 +16.405} C_DIS
 LIN_REL {X  -11.058,Y +7.491,A -0.000,E1 -6.998,E3 +15.775,E4 +15.775} C_DIS
 LIN_REL {X  -26.832,Y +29.974,A -0.000,E1 -20.385,E3 +30.445,E4 +30.445} C_DIS
ENDFOR

HALT
LIN {X -171.253,Y 520.754,Z 0.000,A 30.000, B 0.00, C 0.00,E1 -60.117}
HALT

; PLY 27 OF 41 (Connector)

; ANGLE 51.0 (Not valid for Circ layers and non-tubes)
$APO.CDIS=85
$VEL_EXTAX[1]=100
FOR N_CYC=1 to 1
 LIN_REL {X  +0.000,Y +22.677,A +0.000,E1 -3.946,E3 +12.081,E4 +12.081} C_DIS
 LIN_REL {X  +0.000,Y +6.393,A +0.000,E1 -0.977,E3 +7.230,E4 +7.230} C_DIS
 LIN_REL {X  +0.000,Y -4.768,A +0.000,E1 +0.432,E3 +1.298,E4 +1.298} C_DIS
 LIN_REL {X  +0.000,Y +26.684,A +0.000,E1 -4.019,E3 +6.971,E4 +6.971} C_DIS
 LIN_REL {X  +0.000,Y +9.579,A +0.000,E1 -0.880,E3 +4.554,E4 +4.554} C_DIS
 LIN_REL {X  +0.000,Y +31.423,A +0.000,E1 -1.503,E3 +11.547,E4 +11.547} C_DIS
 LIN_REL {X  +0.000,Y +27.635,A -0.793,E1 -0.168,E3 +12.415,E4 +12.415} C_DIS
 LIN_REL {X  +0.000,Y +22.542,A -6.693,E1 +0.366,E3 +10.125,E4 +10.125} C_DIS
 LIN_REL {X  +0.000,Y +40.084,A -7.603,E1 +0.357,E3 +19.240,E4 +19.240} C_DIS
 LIN_REL {X  +0.000,Y +55.158,A -8.581,E1 +0.783,E3 +29.182,E4 +29.182} C_DIS
 LIN_REL {X  +0.000,Y +66.660,A -5.636,E1 +1.656,E3 +44.970,E4 +44.970} C_DIS
 LIN_REL {X  +0.000,Y +66.114,A -0.688,E1 +3.258,E3 +65.617,E4 +65.617} C_DIS
 LIN_REL {X  +0.000,Y +69.165,A -0.006,E1 +3.732,E3 +77.625,E4 +77.625} C_DIS
 LIN_REL {X  +0.000,Y +71.480,A +0.000,E1 +3.977,E3 +89.154,E4 +89.154} C_DIS
 LIN_REL {X  +0.000,Y +68.255,A -0.000,E1 +4.060,E3 +96.111,E4 +96.111} C_DIS
 LIN_REL {X  +0.000,Y +63.843,A -0.000,E1 +4.158,E3 +102.452,E4 +102.452} C_DIS
 LIN_REL {X  +0.000,Y +58.670,A -0.000,E1 +4.273,E3 +108.259,E4 +108.259} C_DIS
 LIN_REL {X  +0.000,Y +51.432,A -0.014,E1 +4.326,E3 +110.219,E4 +110.219} C_DIS
 LIN_REL {X  +0.000,Y +41.479,A -0.122,E1 +4.305,E3 +103.629,E4 +103.629} C_DIS
 LIN_REL {X  +0.000,Y +29.531,A -0.629,E1 +4.075,E3 +84.895,E4 +84.895} C_DIS
 LIN_REL {X  +0.000,Y +20.296,A -2.558,E1 +3.130,E3 +60.539,E4 +60.539} C_DIS
 LIN_REL {X  +0.000,Y +14.525,A -8.333,E1 +7.611,E3 +48.128,E4 +48.128} C_DIS
 LIN_REL {X  +0.000,Y +7.260,A -11.454,E1 +14.667,E3 +42.881,E4 +42.881} C_DIS
 LIN_REL {X  +0.000,Y +0.268,A -6.203,E1 +11.913,E3 +35.281,E4 +35.281} C_DIS
 LIN_REL {X  +0.000,Y -7.717,A -0.687,E1 +9.636,E3 +43.538,E4 +43.538} C_DIS
 LIN_REL {X  +0.000,Y -9.501,A +0.000,E1 +7.226,E3 +30.819,E4 +30.819} C_DIS
ENDFOR

HALT
LIN {X -166.658,Y 1350.540,Z 0.000,A -30.000, B 0.00, C 0.00,E1 29.993}
HALT

; PLY 28 OF 41 (Helical)

